C09102=1034.938,414.439,357.074,174.357,46.564,159.418
C09103=1034.949,414.684,357.028,174.369,46.569,159.421
C09104=1034.959,414.930,356.980,174.380,46.574,159.424
C09105=1034.970,415.176,356.933,174.392,46.580,159.427
C09106=1034.981,415.420,356.886,174.403,46.585,159.430
C09107=1034.991,415.666,356.839,174.415,46.591,159.433
C09108=1035.002,415.911,356.792,174.426,46.596,159.436
C09109=1035.013,416.157,356.745,174.438,46.602,159.439
C09110=1035.025,416.402,356.697,174.450,46.607,159.441
C09111=1035.035,416.647,356.650,174.461,46.613,159.444
C09112=1035.046,416.893,356.603,174.473,46.618,159.447
C09113=1035.057,417.137,356.555,174.485,46.623,159.450
C09114=1035.068,417.383,356.507,174.497,46.629,159.453
C09115=1035.078,417.628,356.459,174.509,46.635,159.456
C09116=1035.090,417.874,356.412,174.521,46.640,159.459
C09117=1035.100,418.118,356.364,174.533,46.646,159.462
C09118=1035.111,418.364,356.316,174.545,46.651,159.465
C09119=1035.121,418.609,356.269,174.556,46.657,159.468
C09120=1035.132,418.854,356.221,174.568,46.663,159.471
C09121=1035.144,419.100,356.172,174.581,46.668,159.474
C09122=1035.155,419.344,356.125,174.593,46.674,159.477
C09123=1035.166,419.589,356.077,174.605,46.680,159.480
C09124=1035.177,419.835,356.028,174.618,46.685,159.484
C09125=1035.187,420.079,355.980,174.630,46.691,159.487
C09126=1035.199,420.325,355.932,174.642,46.697,159.490
C09127=1035.210,420.570,355.884,174.655,46.703,159.493
C09128=1035.222,420.815,355.836,174.667,46.709,159.496
C09129=1035.233,421.061,355.788,174.679,46.714,159.499
C09130=1035.243,421.305,355.740,174.692,46.720,159.502
C09131=1035.255,421.550,355.691,174.704,46.726,159.506
C09132=1035.266,421.795,355.643,174.717,46.732,159.509
C09133=1035.277,422.041,355.594,174.729,46.738,159.512
C09134=1035.288,422.286,355.545,174.742,46.744,159.515
C09135=1035.300,422.531,355.498,174.754,46.750,159.518
C09136=1035.311,422.775,355.449,174.767,46.756,159.522
C09137=1035.323,423.021,355.400,174.780,46.762,159.525
C09138=1035.334,423.266,355.351,174.793,46.768,159.528
C09139=1035.346,423.511,355.303,174.805,46.774,159.531
C09140=1035.357,423.756,355.254,174.818,46.780,159.535
C09141=1035.368,424.001,355.205,174.832,46.786,159.538
C09142=1035.380,424.246,355.156,174.844,46.792,159.541
C09143=1035.391,424.490,355.107,174.857,46.798,159.545
C09144=1035.403,424.735,355.058,174.871,46.804,159.548
C09145=1035.414,424.982,355.008,174.883,46.810,159.551
C09146=1035.425,425.226,354.959,174.896,46.817,159.555
C09147=1035.437,425.470,354.910,174.910,46.823,159.558
C09148=1035.448,425.715,354.861,174.923,46.829,159.561
C09149=1035.460,425.961,354.811,174.936,46.835,159.565
C09150=1035.471,426.205,354.762,174.949,46.842,159.568
C09151=1035.483,426.450,354.713,174.963,46.848,159.572
C09152=1035.495,426.695,354.663,174.976,46.854,159.575
C09153=1035.507,426.940,354.614,174.990,46.861,159.579
C09154=1035.519,427.185,354.565,175.003,46.867,159.582
C09155=1035.530,427.429,354.515,175.016,46.873,159.585
C09156=1035.542,427.675,354.465,175.030,46.879,159.589
C09157=1035.553,427.919,354.415,175.043,46.886,159.593
C09158=1035.566,428.164,354.365,175.057,46.892,159.596
C09159=1035.577,428.408,354.315,175.071,46.899,159.600
C09160=1035.589,428.654,354.265,175.084,46.905,159.603
C09161=1035.600,428.898,354.216,175.099,46.912,159.607
C09162=1035.612,429.143,354.165,175.113,46.919,159.610
C09163=1035.624,429.387,354.115,175.127,46.925,159.614
C09164=1035.636,429.632,354.065,175.141,46.931,159.618
C09165=1035.647,429.877,354.014,175.154,46.939,159.621
C09166=1035.659,430.121,353.965,175.168,46.945,159.625
C09167=1035.672,430.366,353.915,175.182,46.952,159.629
C09168=1035.683,430.611,353.863,175.196,46.958,159.632
C09169=1035.696,430.855,353.813,175.211,46.965,159.636
C09170=1035.708,431.100,353.763,175.225,46.972,159.640
C09171=1035.719,431.345,353.713,175.239,46.979,159.644
C09172=1035.732,431.589,353.662,175.254,46.985,159.647
C09173=1035.744,431.834,353.612,175.268,46.992,159.651
C09174=1035.757,432.078,353.561,175.282,46.999,159.655
C09175=1035.768,432.323,353.510,175.297,47.005,159.659
C09176=1035.781,432.567,353.459,175.312,47.012,159.663
C09177=1035.793,432.811,353.409,175.326,47.019,159.666
C09178=1035.805,433.057,353.358,175.341,47.026,159.670
C09179=1035.818,433.301,353.307,175.355,47.033,159.674
C09180=1035.830,433.545,353.256,175.371,47.040,159.678
C09181=1035.842,433.789,353.205,175.385,47.047,159.682
C09182=1035.855,434.034,353.154,175.400,47.054,159.686
C09183=1035.867,434.279,353.102,175.415,47.060,159.690
C09184=1035.880,434.523,353.052,175.430,47.068,159.694
C09185=1035.893,434.768,353.000,175.445,47.074,159.697
C09186=1035.905,435.013,352.949,175.460,47.082,159.701
C09187=1035.917,435.257,352.898,175.475,47.089,159.705
C09188=1035.930,435.501,352.846,175.490,47.096,159.709
C09189=1035.942,435.746,352.794,175.505,47.103,159.713
C09190=1035.955,435.990,352.743,175.521,47.110,159.717
C09191=1035.967,436.234,352.691,175.537,47.117,159.721
C09192=1035.980,436.479,352.640,175.552,47.125,159.726
C09193=1035.993,436.725,352.588,175.567,47.132,159.730
C09194=1036.006,436.971,352.535,175.583,47.139,159.734
C09195=1036.018,437.216,352.484,175.598,47.147,159.738
C09196=1036.031,437.462,352.431,175.614,47.154,159.742
C09197=1036.044,437.707,352.379,175.630,47.161,159.746
C09198=1036.057,437.951,352.326,175.646,47.169,159.751
C09199=1036.070,438.195,352.275,175.662,47.176,159.755
C09200=1036.082,438.440,352.222,175.677,47.184,159.759
C09201=1036.095,438.683,352.170,175.693,47.191,159.763
C09202=1036.108,438.928,352.118,175.709,47.198,159.767
C09203=1036.121,439.172,352.066,175.725,47.206,159.772
C09204=1036.134,439.417,352.013,175.741,47.214,159.776
C09205=1036.147,439.660,351.961,175.757,47.221,159.780
C09206=1036.160,439.904,351.909,175.773,47.228,159.785
C09207=1036.173,440.148,351.855,175.789,47.236,159.789
C09208=1036.186,440.393,351.804,175.807,47.243,159.793
C09209=1036.199,440.637,351.750,175.823,47.251,159.798
C09210=1036.212,440.881,351.698,175.839,47.259,159.802
C09211=1036.225,441.125,351.645,175.856,47.267,159.807
C09212=1036.238,441.369,351.592,175.872,47.274,159.811
C09213=1036.252,441.613,351.539,175.889,47.282,159.816
C09214=1036.265,441.857,351.486,175.906,47.290,159.820
C09215=1036.278,442.101,351.432,175.922,47.297,159.825
C09216=1036.292,442.345,351.379,175.940,47.305,159.829
C09217=1036.305,442.588,351.327,175.956,47.313,159.834
C09218=1036.319,442.832,351.273,175.973,47.320,159.838
C09219=1036.332,443.076,351.220,175.990,47.329,159.843
C09220=1036.345,443.320,351.167,176.008,47.336,159.847
C09221=1036.359,443.563,351.114,176.024,47.344,159.852
C09222=1036.372,443.807,351.061,176.042,47.352,159.857
C09223=1036.386,444.050,351.007,176.058,47.360,159.861
C09224=1036.399,444.294,350.954,176.076,47.368,159.866
C09225=1036.414,444.537,350.901,176.094,47.376,159.870
C09226=1036.429,444.780,350.850,176.111,47.384,159.875
C09227=1036.445,445.024,350.797,176.129,47.391,159.880
C09228=1036.461,445.267,350.746,176.146,47.399,159.884
C09229=1036.478,445.511,350.695,176.164,47.406,159.889
C09230=1036.495,445.755,350.645,176.182,47.413,159.893
C09231=1036.513,445.999,350.595,176.200,47.421,159.898
C09232=1036.531,446.243,350.545,176.218,47.428,159.903
C09233=1036.550,446.486,350.497,176.236,47.435,159.907
C09234=1036.569,446.731,350.447,176.254,47.442,159.911
C09235=1036.589,446.975,350.399,176.272,47.449,159.916
C09236=1036.609,447.220,350.351,176.291,47.456,159.921
C09237=1036.630,447.464,350.304,176.309,47.462,159.925
C09238=1036.652,447.708,350.257,176.327,47.469,159.929
C09239=1036.673,447.953,350.211,176.346,47.475,159.934
C09240=1036.697,448.198,350.165,176.364,47.482,159.938
C09241=1036.719,448.442,350.119,176.383,47.488,159.943
C09242=1036.743,448.687,350.074,176.401,47.495,159.947
C09243=1036.767,448.931,350.029,176.421,47.501,159.952
C09244=1036.792,449.177,349.985,176.440,47.507,159.956
C09245=1036.817,449.422,349.941,176.459,47.513,159.961
C09246=1036.843,449.667,349.898,176.478,47.519,159.965
C09247=1036.869,449.912,349.855,176.497,47.525,159.969
C09248=1036.896,450.157,349.812,176.517,47.530,159.974
C09249=1036.924,450.403,349.771,176.536,47.536,159.978
C09250=1036.951,450.649,349.729,176.555,47.541,159.982
C09251=1036.980,450.893,349.687,176.575,47.548,159.987
C09252=1037.009,451.139,349.647,176.594,47.553,159.991
C09253=1037.046,451.441,349.597,176.619,47.560,159.996
C09254=1037.083,451.744,349.549,176.644,47.566,160.002
C09255=1037.122,452.046,349.501,176.668,47.572,160.007
C09256=1037.160,452.347,349.453,176.693,47.578,160.012
C09257=1036.869,452.403,349.129,176.696,47.649,160.034
C09258=1036.832,452.115,349.174,176.672,47.644,160.029
C09259=1036.796,451.826,349.221,176.648,47.637,160.024
C09260=1036.760,451.537,349.267,176.625,47.632,160.019
C09261=1036.724,451.248,349.314,176.602,47.626,160.014
C09262=1036.695,451.003,349.354,176.582,47.620,160.010
C09263=1036.666,450.758,349.395,176.562,47.615,160.006
C09264=1036.638,450.512,349.436,176.543,47.609,160.001
C09265=1036.610,450.266,349.478,176.523,47.604,159.997
C09266=1036.583,450.021,349.520,176.504,47.598,159.992
C09267=1036.557,449.776,349.563,176.484,47.592,159.988
C09268=1036.531,449.531,349.606,176.465,47.586,159.984
C09269=1036.504,449.286,349.650,176.446,47.580,159.979
C09270=1036.480,449.041,349.693,176.427,47.574,159.975
C09271=1036.455,448.796,349.739,176.408,47.569,159.971
C09272=1036.431,448.551,349.783,176.389,47.562,159.966
C09273=1036.407,448.306,349.829,176.371,47.556,159.962
C09274=1036.385,448.062,349.874,176.351,47.549,159.957
C09275=1036.363,447.816,349.920,176.333,47.543,159.953
C09276=1036.341,447.572,349.967,176.314,47.537,159.948
C09277=1036.319,447.328,350.014,176.296,47.530,159.944
C09278=1036.298,447.084,350.062,176.278,47.523,159.939
C09279=1036.279,446.839,350.110,176.259,47.517,159.935
C09280=1036.259,446.595,350.159,176.241,47.510,159.930
C09281=1036.240,446.351,350.206,176.223,47.503,159.926
C09282=1036.221,446.107,350.256,176.204,47.496,159.921
C09283=1036.203,445.863,350.306,176.187,47.489,159.917
C09284=1036.185,445.619,350.356,176.168,47.482,159.912
C09285=1036.169,445.375,350.407,176.151,47.474,159.908
C09286=1036.152,445.132,350.458,176.133,47.467,159.903
C09287=1036.137,444.888,350.509,176.116,47.459,159.898
C09288=1036.121,444.645,350.561,176.098,47.452,159.894
C09289=1036.106,444.402,350.613,176.081,47.444,159.889
C09290=1036.092,444.159,350.667,176.063,47.437,159.885
C09291=1036.078,443.915,350.719,176.046,47.429,159.880
C09292=1036.065,443.672,350.773,176.029,47.421,159.875
C09293=1036.051,443.429,350.827,176.011,47.413,159.871
C09294=1036.038,443.185,350.880,175.994,47.405,159.866
C09295=1036.025,442.941,350.933,175.977,47.398,159.862
C09296=1036.011,442.697,350.986,175.960,47.390,159.857
C09297=1035.997,442.453,351.039,175.943,47.382,159.852
C09298=1035.984,442.209,351.093,175.926,47.375,159.848
C09299=1035.970,441.966,351.146,175.910,47.367,159.843
C09300=1035.957,441.721,351.198,175.892,47.359,159.839
C09301=1035.944,441.477,351.251,175.876,47.351,159.834
C09302=1035.931,441.233,351.305,175.859,47.344,159.830
C09303=1035.917,440.989,351.357,175.842,47.336,159.825
C09304=1035.904,440.745,351.410,175.826,47.328,159.821
C09305=1035.891,440.501,351.463,175.809,47.321,159.817
C09306=1035.878,440.257,351.516,175.793,47.314,159.812
C09307=1035.866,440.013,351.568,175.777,47.306,159.808
C09308=1035.852,439.769,351.621,175.761,47.298,159.804
C09309=1035.839,439.525,351.673,175.744,47.291,159.799
C09310=1035.826,439.281,351.727,175.728,47.284,159.795
C09311=1035.813,439.036,351.778,175.711,47.276,159.791
C09312=1035.800,438.793,351.831,175.695,47.269,159.786
C09313=1035.787,438.548,351.882,175.679,47.262,159.782
C09314=1035.774,438.304,351.935,175.664,47.255,159.778
C09315=1035.762,438.060,351.987,175.648,47.247,159.774
C09316=1035.748,437.815,352.039,175.632,47.239,159.769
C09317=1035.736,437.571,352.091,175.617,47.233,159.765
C09318=1035.723,437.324,352.145,175.600,47.225,159.761
C09319=1035.710,437.076,352.197,175.584,47.218,159.757
C09320=1035.697,436.829,352.249,175.569,47.211,159.753
C09321=1035.684,436.582,352.302,175.553,47.203,159.749
C09322=1035.672,436.338,352.353,175.538,47.196,159.745
C09323=1035.659,436.094,352.405,175.522,47.189,159.740
C09324=1035.646,435.849,352.457,175.506,47.182,159.736
C09325=1035.634,435.605,352.508,175.492,47.175,159.732
C09326=1035.622,435.361,352.559,175.476,47.168,159.728
C09327=1035.608,435.116,352.611,175.461,47.161,159.724
C09328=1035.596,434.872,352.663,175.446,47.154,159.720
C09329=1035.584,434.628,352.714,175.431,47.147,159.716
C09330=1035.572,434.383,352.765,175.415,47.140,159.712
C09331=1035.559,434.138,352.816,175.401,47.133,159.709
C09332=1035.547,433.894,352.868,175.387,47.126,159.705
C09333=1035.534,433.650,352.918,175.371,47.119,159.701
C09334=1035.522,433.405,352.968,175.356,47.112,159.697
C09335=1035.510,433.160,353.020,175.341,47.106,159.693
C09336=1035.497,432.915,353.071,175.326,47.099,159.689
C09337=1035.484,432.671,353.122,175.312,47.092,159.685
C09338=1035.472,432.426,353.173,175.298,47.085,159.681
C09339=1035.460,432.182,353.223,175.283,47.078,159.678
C09340=1035.447,431.938,353.274,175.268,47.072,159.674
C09341=1035.435,431.694,353.324,175.254,47.065,159.670
C09342=1035.424,431.448,353.375,175.239,47.059,159.666
C09343=1035.411,431.204,353.425,175.225,47.052,159.663
C09344=1035.399,430.959,353.476,175.211,47.045,159.659
C09345=1035.387,430.714,353.526,175.197,47.039,159.655
C09346=1035.375,430.470,353.577,175.182,47.032,159.651
C09347=1035.363,430.226,353.627,175.168,47.025,159.648
C09348=1035.351,429.981,353.677,175.154,47.019,159.644
C09349=1035.339,429.736,353.728,175.140,47.012,159.641
C09350=1035.327,429.491,353.778,175.126,47.006,159.637
C09351=1035.316,429.247,353.828,175.112,47.000,159.633
C09352=1035.304,429.002,353.878,175.098,46.992,159.630
C09353=1035.292,428.758,353.928,175.084,46.986,159.626
C09354=1035.280,428.513,353.978,175.070,46.980,159.622
C09355=1035.269,428.268,354.028,175.056,46.973,159.619
C09356=1035.257,428.023,354.078,175.042,46.967,159.615
C09357=1035.245,427.779,354.127,175.029,46.960,159.612
C09358=1035.233,427.534,354.178,175.016,46.955,159.608
C09359=1035.222,427.289,354.227,175.002,46.948,159.605
C09360=1035.210,427.044,354.277,174.989,46.942,159.601
C09361=1035.198,426.799,354.326,174.975,46.936,159.598
C09362=1035.186,426.554,354.375,174.961,46.929,159.594
C09363=1035.174,426.310,354.425,174.948,46.923,159.591
C09364=1035.162,426.064,354.475,174.934,46.917,159.587
C09365=1035.151,425.820,354.524,174.921,46.911,159.584
C09366=1035.140,425.575,354.573,174.907,46.904,159.581
C09367=1035.128,425.329,354.623,174.895,46.898,159.577
C09368=1035.117,425.085,354.672,174.881,46.892,159.574
C09369=1035.105,424.840,354.721,174.868,46.886,159.571
C09370=1035.094,424.596,354.770,174.856,46.880,159.567
C09371=1035.083,424.350,354.819,174.842,46.874,159.564
C09372=1035.071,424.105,354.868,174.829,46.868,159.561
C09373=1035.059,423.860,354.917,174.816,46.862,159.557
C09374=1035.048,423.615,354.966,174.803,46.856,159.554
C09375=1035.037,423.371,355.015,174.790,46.850,159.551
C09376=1035.025,423.125,355.063,174.778,46.844,159.548
C09377=1035.014,422.880,355.112,174.764,46.838,159.544
C09378=1035.003,422.633,355.161,174.752,46.832,159.541
C09379=1034.990,422.386,355.210,174.739,46.826,159.538
C09380=1034.979,422.138,355.259,174.726,46.821,159.534
C09381=1034.968,421.890,355.308,174.713,46.814,159.531
C09382=1034.957,421.645,355.356,174.701,46.809,159.528
C09383=1034.945,421.400,355.405,174.688,46.803,159.525
C09384=1034.934,421.155,355.453,174.676,46.797,159.522
C09385=1034.923,420.910,355.501,174.663,46.791,159.519
C09386=1034.912,420.665,355.549,174.651,46.786,159.515
C09387=1034.901,420.421,355.598,174.639,46.780,159.512
C09388=1034.890,420.175,355.647,174.626,46.774,159.509
C09389=1034.878,419.930,355.695,174.614,46.769,159.506
C09390=1034.867,419.685,355.742,174.602,46.763,159.503
C09391=1034.856,419.440,355.791,174.590,46.757,159.500
C09392=1034.845,419.194,355.838,174.577,46.752,159.497
C09393=1034.834,418.949,355.887,174.565,46.746,159.494
C09394=1034.824,418.704,355.934,174.553,46.740,159.491
C09395=1034.813,418.459,355.983,174.541,46.735,159.488
C09396=1034.801,418.214,356.030,174.528,46.729,159.485
C09397=1034.791,417.968,356.078,174.517,46.723,159.482
C09398=1034.780,417.724,356.126,174.505,46.718,159.479
C09399=1034.769,417.478,356.174,174.493,46.712,159.476
C09400=1034.759,417.233,356.221,174.481,46.707,159.473
C09401=1034.747,416.988,356.269,174.468,46.702,159.470
C09402=1034.737,416.743,356.316,174.457,46.696,159.467
C09403=1034.725,416.497,356.363,174.445,46.691,159.464
C09404=1034.715,416.252,356.411,174.433,46.686,159.461
C09405=1034.703,416.007,356.458,174.422,46.680,159.458
C09406=1034.693,415.761,356.505,174.410,46.675,159.455
C09407=1034.682,415.515,356.553,174.398,46.669,159.452
C09408=1034.671,415.271,356.599,174.387,46.664,159.449
C09409=1034.661,415.025,356.647,174.375,46.659,159.446
C09410=1034.650,414.780,356.694,174.363,46.654,159.444
C09411=1034.639,414.535,356.741,174.352,46.648,159.441
C09412=1034.628,414.289,356.787,174.340,46.643,159.438
C09413=1034.618,414.044,356.835,174.330,46.638,159.435
C09414=1034.607,413.799,356.881,174.318,46.633,159.432
C09415=1034.597,413.553,356.929,174.307,46.627,159.430
C09416=1034.586,413.308,356.975,174.295,46.623,159.427
C09417=1034.575,413.063,357.023,174.284,46.617,159.424
C09418=1034.566,412.817,357.069,174.272,46.612,159.421
C09419=1034.555,412.572,357.116,174.261,46.607,159.419
C09420=1034.544,412.327,357.163,174.250,46.602,159.416
C09421=1034.534,412.081,357.209,174.239,46.597,159.413
C09422=1034.524,411.836,357.256,174.228,46.591,159.410
C09423=1034.513,411.590,357.302,174.217,46.586,159.408
C09424=1034.503,411.345,357.349,174.205,46.582,159.405
C09425=1034.492,411.099,357.395,174.194,46.576,159.402
C09426=1034.482,410.854,357.442,174.184,46.571,159.399
C09427=1034.471,410.608,357.488,174.172,46.567,159.397
C09428=1034.461,410.363,357.534,174.162,46.562,159.394
C09429=1034.450,410.117,357.580,174.151,46.557,159.391
C09430=1034.440,409.871,357.627,174.140,46.552,159.389
C09431=1034.430,409.626,357.672,174.129,46.547,159.386
C09432=1034.419,409.381,357.719,174.118,46.542,159.384
C09433=1034.408,409.135,357.765,174.108,46.538,159.381
C09434=1034.398,408.893,357.810,174.097,46.533,159.378
C09435=1034.389,408.651,357.855,174.086,46.528,159.376
C09436=1034.378,408.410,357.900,174.076,46.523,159.373
C09437=1034.367,408.168,357.946,174.065,46.518,159.371
C09438=1034.358,407.926,357.990,174.055,46.514,159.368
C09439=1034.347,407.685,358.036,174.044,46.509,159.366
C09440=1034.338,407.443,358.081,174.034,46.504,159.363
C09441=1034.328,407.201,358.126,174.024,46.500,159.361
C09442=1034.317,406.955,358.172,174.013,46.495,159.358
C09443=1034.308,406.710,358.216,174.003,46.491,159.356
C09444=1034.297,406.464,358.262,173.992,46.486,159.353
C09445=1034.287,406.219,358.308,173.982,46.481,159.351
C09446=1034.277,405.973,358.354,173.972,46.477,159.348
C09447=1034.267,405.728,358.399,173.961,46.472,159.346
C09448=1034.257,405.482,358.444,173.951,46.467,159.343
C09449=1034.247,405.237,358.490,173.940,46.463,159.341
C09450=1034.237,404.991,358.535,173.930,46.458,159.339
C09451=1034.228,404.745,358.581,173.920,46.454,159.336
C09452=1034.217,404.499,358.626,173.909,46.449,159.333
C09453=1034.207,404.254,358.671,173.900,46.444,159.331
C09454=1034.198,404.008,358.716,173.889,46.440,159.329
C09455=1034.187,403.763,358.762,173.879,46.435,159.326
C09456=1034.177,403.517,358.807,173.869,46.431,159.324
C09457=1034.168,403.271,358.852,173.859,46.427,159.322
C09458=1034.158,403.025,358.897,173.850,46.422,159.319
C09459=1034.148,402.779,358.942,173.839,46.418,159.317
C09460=1034.139,402.534,358.987,173.829,46.413,159.314
C09461=1034.129,402.288,359.032,173.819,46.409,159.312
C09462=1034.118,402.042,359.077,173.809,46.405,159.310
C09463=1034.109,401.797,359.122,173.799,46.400,159.307
C09464=1034.099,401.551,359.167,173.789,46.395,159.305
C09465=1034.089,401.306,359.212,173.779,46.391,159.303
C09466=1034.080,401.060,359.256,173.770,46.387,159.300
C09467=1034.070,400.814,359.301,173.760,46.383,159.298
C09468=1034.060,400.568,359.346,173.749,46.378,159.296
C09469=1034.050,400.322,359.390,173.740,46.374,159.294
C09470=1034.040,400.077,359.434,173.730,46.370,159.291
C09471=1034.030,399.831,359.479,173.720,46.366,159.289
C09472=1034.021,399.585,359.523,173.711,46.361,159.287
C09473=1034.011,399.339,359.568,173.701,46.358,159.285
C09474=1034.002,399.093,359.612,173.692,46.353,159.282
C09475=1033.992,398.847,359.656,173.682,46.349,159.280
C09476=1033.982,398.602,359.700,173.672,46.345,159.278
C09477=1033.973,398.356,359.744,173.663,46.341,159.276
C09478=1033.963,398.110,359.788,173.653,46.337,159.273
C09479=1033.953,397.864,359.833,173.644,46.332,159.271
C09480=1033.944,397.619,359.876,173.634,46.328,159.269
C09481=1033.934,397.373,359.921,173.625,46.324,159.267
C09482=1033.925,397.145,359.962,173.616,46.321,159.265
C09483=1033.917,396.916,360.002,173.608,46.317,159.263
C09484=1033.908,396.687,360.044,173.599,46.313,159.261
C09485=1033.899,396.460,360.084,173.590,46.310,159.259
C09486=1033.890,396.231,360.124,173.582,46.306,159.257
C09487=1033.881,396.003,360.166,173.573,46.302,159.255
C09488=1033.873,395.775,360.207,173.564,46.299,159.253
C09489=1033.863,395.546,360.246,173.556,46.295,159.251
C09490=1033.854,395.300,360.291,173.547,46.291,159.249
C09491=1033.845,395.055,360.334,173.537,46.287,159.247
C09492=1033.836,394.809,360.378,173.528,46.283,159.245
C09493=1033.826,394.563,360.422,173.519,46.279,159.243
C09494=1033.817,394.317,360.465,173.509,46.276,159.241
C09495=1033.808,394.071,360.509,173.500,46.271,159.238
C09496=1033.798,393.825,360.553,173.492,46.268,159.236
C09497=1033.789,393.579,360.596,173.482,46.264,159.234
C09498=1033.779,393.327,360.641,173.473,46.260,159.232
C09499=1033.769,393.074,360.685,173.463,46.256,159.230
C09500=1033.760,392.822,360.729,173.454,46.252,159.228
C09501=1033.750,392.570,360.774,173.445,46.248,159.226
C09502=1033.741,392.324,360.817,173.436,46.245,159.224
C09503=1033.732,392.078,360.860,173.427,46.241,159.222
C09504=1033.722,391.832,360.903,173.419,46.237,159.220
C09505=1033.713,391.586,360.947,173.410,46.233,159.218
C09506=1033.704,391.340,360.989,173.400,46.230,159.216
C09507=1033.695,391.093,361.033,173.391,46.226,159.214
C09508=1033.685,390.848,361.076,173.383,46.222,159.212
C09509=1033.677,390.602,361.119,173.374,46.218,159.210
C09510=1033.667,390.356,361.162,173.365,46.215,159.208
C09511=1033.658,390.110,361.205,173.357,46.212,159.206
C09512=1033.648,389.863,361.247,173.347,46.208,159.204
C09513=1033.639,389.617,361.290,173.339,46.204,159.202
C09514=1033.631,389.371,361.333,173.330,46.201,159.200
C09515=1033.621,389.125,361.376,173.321,46.197,159.198
C09516=1033.612,388.879,361.419,173.313,46.194,159.197
C09517=1033.603,388.633,361.461,173.304,46.190,159.195
C09518=1033.594,388.387,361.504,173.296,46.186,159.193
C09519=1033.585,388.141,361.547,173.287,46.183,159.191
C09520=1033.575,387.895,361.589,173.279,46.180,159.189
C09521=1033.567,387.648,361.631,173.270,46.176,159.187
C09522=1033.558,387.402,361.674,173.262,46.173,159.185
C09523=1033.548,387.156,361.717,173.253,46.169,159.183
C09524=1033.539,386.910,361.759,173.245,46.166,159.181
C09525=1033.530,386.664,361.801,173.236,46.162,159.179
C09526=1033.521,386.418,361.844,173.228,46.159,159.178
C09527=1033.512,386.172,361.885,173.219,46.156,159.176
C09528=1033.503,385.925,361.929,173.211,46.152,159.174
C09529=1033.494,385.679,361.970,173.202,46.149,159.172
C09530=1033.485,385.433,362.013,173.194,46.146,159.170
C09531=1033.476,385.187,362.055,173.186,46.143,159.169
C09532=1033.467,384.940,362.096,173.177,46.139,159.167
C09533=1033.457,384.694,362.139,173.169,46.136,159.165
C09534=1033.449,384.448,362.180,173.160,46.132,159.163
C09535=1033.440,384.202,362.222,173.152,46.129,159.161
C09536=1033.431,383.955,362.264,173.144,46.126,159.160
C09537=1033.421,383.710,362.306,173.135,46.123,159.158
C09538=1033.412,383.463,362.348,173.128,46.120,159.156
C09539=1033.404,383.217,362.390,173.120,46.116,159.154
C09540=1033.395,382.970,362.432,173.111,46.113,159.153
C09541=1033.386,382.724,362.474,173.103,46.110,159.151
C09542=1033.377,382.477,362.515,173.095,46.107,159.149
C09543=1033.369,382.231,362.557,173.086,46.104,159.147
C09544=1033.360,381.985,362.599,173.079,46.100,159.146
C09545=1033.351,381.738,362.641,173.070,46.097,159.144
C09546=1033.342,381.493,362.682,173.062,46.094,159.142
C09547=1033.333,381.246,362.724,173.054,46.091,159.140
C09548=1033.324,381.000,362.765,173.046,46.088,159.139
C09549=1033.316,380.754,362.807,173.038,46.085,159.137
C09550=1033.307,380.507,362.849,173.030,46.082,159.135
C09551=1033.298,380.261,362.891,173.022,46.079,159.134
C09552=1033.289,380.015,362.932,173.015,46.075,159.132
C09553=1033.281,379.768,362.973,173.006,46.072,159.130
C09554=1033.274,379.554,363.009,173.000,46.070,159.129
C09555=1033.266,379.341,363.045,172.993,46.067,159.127
C09556=1033.259,379.126,363.082,172.986,46.065,159.126
C09557=1033.251,378.912,363.117,172.979,46.062,159.124
C09558=1033.244,378.698,363.153,172.972,46.060,159.123
C09559=1033.236,378.484,363.189,172.965,46.057,159.122
C09560=1033.229,378.270,363.226,172.958,46.055,159.120
C09561=1033.221,378.056,363.261,172.952,46.051,159.119
C09562=1033.213,377.810,363.302,172.944,46.049,159.117
C09563=1033.204,377.563,363.343,172.936,46.046,159.115
C09564=1033.196,377.316,363.384,172.929,46.043,159.114
C09565=1033.187,377.071,363.425,172.921,46.040,159.112
C09566=1033.178,376.824,363.466,172.913,46.038,159.111
C09567=1033.169,376.577,363.507,172.905,46.034,159.109
C09568=1033.161,376.331,363.548,172.897,46.031,159.107
C09569=1033.152,376.085,363.589,172.890,46.029,159.106
C09570=1033.144,375.838,363.629,172.882,46.026,159.104
C09571=1033.135,375.591,363.670,172.874,46.023,159.103
C09572=1033.126,375.345,363.710,172.867,46.020,159.101
C09573=1033.118,375.098,363.751,172.859,46.018,159.100
C09574=1033.110,374.852,363.792,172.852,46.015,159.098
C09575=1033.101,374.606,363.834,172.844,46.012,159.097
C09576=1033.092,374.360,363.874,172.837,46.009,159.095
C09577=1033.083,374.113,363.915,172.829,46.007,159.094
C09578=1033.075,373.867,363.956,172.822,46.004,159.092
C09579=1033.066,373.620,363.996,172.814,46.001,159.090
C09580=1033.058,373.373,364.036,172.807,45.998,159.089
C09581=1033.050,373.127,364.076,172.799,45.996,159.087
C09582=1033.041,372.880,364.117,172.792,45.993,159.086
C09583=1033.033,372.634,364.158,172.784,45.990,159.084
C09584=1033.024,372.387,364.199,172.777,45.987,159.083
C09585=1033.016,372.140,364.239,172.769,45.985,159.081
C09586=1033.008,371.894,364.278,172.762,45.982,159.080
C09587=1032.999,371.647,364.319,172.755,45.979,159.078
C09588=1032.991,371.401,364.360,172.747,45.977,159.077
C09589=1032.982,371.155,364.400,172.740,45.974,159.075
C09590=1032.974,370.908,364.440,172.732,45.972,159.074
C09591=1032.966,370.661,364.481,172.725,45.969,159.072
C09592=1032.958,370.414,364.522,172.718,45.967,159.071
C09593=1032.949,370.168,364.561,172.710,45.964,159.069
C09594=1032.941,369.922,364.602,172.704,45.962,159.068
C09595=1032.934,369.675,364.642,172.697,45.959,159.067
C09596=1032.924,369.428,364.682,172.689,45.957,159.065
C09597=1032.916,369.181,364.722,172.682,45.954,159.064
C09598=1032.908,368.935,364.761,172.675,45.951,159.062
C09599=1032.899,368.689,364.801,172.667,45.949,159.061
C09600=1032.892,368.442,364.841,172.660,45.946,159.059
C09601=1032.882,368.194,364.881,172.654,45.944,159.058
C09602=1032.874,367.948,364.920,172.646,45.942,159.057
C09603=1032.866,367.701,364.961,172.639,45.939,159.055
C09604=1032.858,367.455,365.000,172.632,45.937,159.054
C09605=1032.849,367.208,365.039,172.624,45.935,159.052
C09606=1032.841,366.961,365.079,172.618,45.932,159.051
C09607=1032.833,366.715,365.119,172.611,45.929,159.050
C09608=1032.825,366.468,365.159,172.604,45.927,159.048
C09609=1032.817,366.221,365.198,172.596,45.925,159.047
C09610=1032.808,365.975,365.238,172.590,45.923,159.046
C09611=1032.800,365.728,365.278,172.583,45.920,159.044
C09612=1032.792,365.482,365.317,172.576,45.918,159.043
C09613=1032.784,365.235,365.356,172.568,45.916,159.041
C09614=1032.770,364.828,365.422,172.557,45.912,159.039
C09615=1032.756,364.420,365.487,172.546,45.908,159.037
C09616=1032.743,364.013,365.552,172.535,45.904,159.035
C09617=1032.730,363.606,365.617,172.523,45.900,159.033
C09618=1032.722,363.359,365.656,172.516,45.898,159.031
C09619=1032.713,363.113,365.695,172.510,45.896,159.030
C09620=1032.706,362.865,365.735,172.503,45.894,159.029
C09621=1032.697,362.618,365.774,172.496,45.892,159.027
C09622=1032.690,362.373,365.813,172.488,45.890,159.026
C09623=1032.682,362.125,365.852,172.482,45.887,159.025
C09624=1032.674,361.878,365.891,172.475,45.885,159.023
C09625=1032.665,361.632,365.931,172.469,45.883,159.022
C09626=1032.658,361.384,365.970,172.462,45.881,159.021
C09627=1032.650,361.138,366.009,172.455,45.878,159.020
C09628=1032.642,360.891,366.048,172.449,45.877,159.018
C09629=1032.633,360.645,366.087,172.442,45.874,159.017
C09630=1032.625,360.397,366.125,172.435,45.872,159.016
C09631=1032.618,360.151,366.164,172.429,45.870,159.015
C09632=1032.609,359.904,366.203,172.422,45.868,159.013
C09633=1032.601,359.657,366.242,172.415,45.866,159.012
C09634=1032.594,359.410,366.281,172.408,45.864,159.011
C09635=1032.586,359.164,366.320,172.401,45.862,159.010
C09636=1032.578,358.916,366.358,172.395,45.860,159.008
C09637=1032.569,358.669,366.397,172.388,45.858,159.007
C09638=1032.562,358.423,366.435,172.382,45.856,159.006
C09639=1032.553,358.176,366.475,172.375,45.854,159.005
C09640=1032.545,357.929,366.513,172.369,45.852,159.004
C09641=1032.538,357.682,366.551,172.362,45.850,159.002
C09642=1032.530,357.435,366.590,172.356,45.848,159.001
C09643=1032.521,357.188,366.629,172.349,45.846,159.000
C09644=1032.514,356.941,366.667,172.342,45.844,158.999
C09645=1032.506,356.694,366.706,172.336,45.842,158.997
C09646=1032.498,356.448,366.744,172.329,45.840,158.996
C09647=1032.490,356.200,366.782,172.323,45.839,158.995
C09648=1032.483,355.954,366.821,172.316,45.836,158.994
C09649=1032.474,355.707,366.859,172.310,45.834,158.993
C09650=1032.466,355.460,366.898,172.303,45.833,158.992
C09651=1032.459,355.213,366.936,172.297,45.831,158.990
C09652=1032.450,354.965,366.973,172.292,45.829,158.989
C09653=1032.443,354.719,367.012,172.285,45.827,158.988
C09654=1032.434,354.472,367.050,172.279,45.825,158.987
C09655=1032.427,354.225,367.088,172.272,45.824,158.986
C09656=1032.419,353.977,367.126,172.266,45.822,158.985
C09657=1032.411,353.731,367.164,172.259,45.820,158.984
C09658=1032.403,353.484,367.203,172.253,45.818,158.982
C09659=1032.395,353.237,367.240,172.247,45.816,158.981
C09660=1032.388,352.990,367.278,172.240,45.815,158.980
C09661=1032.380,352.743,367.317,172.234,45.813,158.979
C09662=1032.372,352.496,367.354,172.227,45.811,158.978
C09663=1032.363,352.249,367.393,172.222,45.809,158.977
C09664=1032.356,352.002,367.430,172.215,45.807,158.976
C09665=1032.349,351.755,367.468,172.209,45.806,158.974
C09666=1032.341,351.508,367.506,172.203,45.804,158.973
C09667=1032.333,351.261,367.544,172.196,45.803,158.972
C09668=1032.325,351.014,367.581,172.190,45.801,158.971
C09669=1032.317,350.767,367.620,172.185,45.799,158.970
C09670=1032.305,350.366,367.681,172.174,45.796,158.968
C09671=1032.293,349.965,367.742,172.164,45.794,158.967
C09672=1032.279,349.564,367.803,172.154,45.791,158.965
C09673=1032.267,349.163,367.865,172.144,45.788,158.963
C09674=1032.260,348.916,367.902,172.138,45.786,158.962
C09675=1032.253,348.669,367.940,172.132,45.785,158.961
C09676=1032.244,348.422,367.978,172.126,45.783,158.960
C09677=1032.237,348.175,368.015,172.119,45.782,158.959
C09678=1032.229,347.928,368.052,172.113,45.780,158.958
C09679=1032.221,347.681,368.090,172.108,45.778,158.957
C09680=1032.213,347.434,368.127,172.102,45.777,158.956
C09681=1032.206,347.186,368.164,172.095,45.775,158.955
C09682=1032.198,346.940,368.201,172.089,45.774,158.954
C09683=1032.190,346.692,368.239,172.084,45.772,158.953
C09684=1032.182,346.446,368.276,172.078,45.771,158.952
C09685=1032.175,346.198,368.313,172.071,45.769,158.950
C09686=1032.167,345.952,368.350,172.066,45.768,158.950
C09687=1032.160,345.705,368.388,172.060,45.767,158.949
C09688=1032.152,345.458,368.425,172.053,45.765,158.947
C09689=1032.144,345.209,368.462,172.047,45.764,158.946
C09690=1032.136,344.962,368.499,172.042,45.762,158.946
C09691=1032.129,344.715,368.536,172.036,45.760,158.944
C09692=1032.121,344.468,368.573,172.030,45.759,158.943
C09693=1032.114,344.221,368.611,172.024,45.758,158.943
C09694=1032.106,343.974,368.647,172.018,45.756,158.942
C09695=1032.099,343.727,368.685,172.012,45.755,158.940
C09696=1032.091,343.480,368.722,172.007,45.753,158.940
C09697=1032.084,343.232,368.758,172.001,45.752,158.939
C09698=1032.076,342.985,368.795,171.994,45.751,158.938
C09699=1032.069,342.738,368.833,171.989,45.749,158.937
C09700=1032.061,342.491,368.869,171.983,45.747,158.936
C09701=1032.053,342.244,368.906,171.977,45.746,158.935
C09702=1032.046,341.997,368.943,171.972,45.745,158.934
C09703=1032.038,341.749,368.980,171.965,45.744,158.933
C09704=1032.032,341.503,369.017,171.960,45.742,158.932
C09705=1032.024,341.255,369.053,171.954,45.741,158.931
C09706=1032.016,341.009,369.090,171.948,45.740,158.930
C09707=1032.009,340.761,369.127,171.943,45.738,158.929
C09708=1032.001,340.513,369.163,171.937,45.737,158.928
C09709=1031.993,340.267,369.200,171.932,45.736,158.927
C09710=1031.986,340.019,369.236,171.925,45.734,158.926
C09711=1031.979,339.771,369.273,171.919,45.733,158.925
C09712=1031.971,339.525,369.310,171.914,45.732,158.924
C09713=1031.964,339.278,369.346,171.908,45.730,158.923
C09714=1031.956,339.030,369.382,171.903,45.730,158.923
C09715=1031.948,338.783,369.418,171.897,45.728,158.922
C09716=1031.940,338.536,369.455,171.891,45.727,158.921
C09717=1031.933,338.288,369.492,171.886,45.726,158.920
C09718=1031.926,338.041,369.528,171.880,45.725,158.919
C09719=1031.919,337.794,369.564,171.875,45.724,158.918
C09720=1031.911,337.547,369.600,171.869,45.722,158.917
C09721=1031.903,337.299,369.636,171.863,45.721,158.916
C09722=1031.895,337.052,369.673,171.857,45.720,158.915
C09723=1031.889,336.805,369.710,171.852,45.719,158.914
C09724=1031.881,336.558,369.746,171.846,45.718,158.913
C09725=1031.874,336.311,369.782,171.841,45.716,158.913
C09726=1031.862,335.906,369.841,171.831,45.715,158.911
C09727=1031.850,335.502,369.901,171.823,45.713,158.910
C09728=1031.838,335.098,369.960,171.814,45.711,158.908
C09729=1031.826,334.694,370.019,171.804,45.709,158.907
C09730=1031.819,334.446,370.055,171.799,45.708,158.906
C09731=1031.811,334.199,370.091,171.793,45.707,158.905
C09732=1031.804,333.952,370.127,171.788,45.706,158.904
C09733=1031.796,333.704,370.162,171.782,45.705,158.903
C09734=1031.789,333.457,370.198,171.777,45.704,158.903
C09735=1031.781,333.210,370.234,171.771,45.703,158.902
C09736=1031.774,332.962,370.269,171.766,45.702,158.901
C09737=1031.766,332.715,370.305,171.762,45.701,158.900
C09738=1031.759,332.468,370.341,171.755,45.700,158.899
C09739=1031.752,332.220,370.376,171.751,45.699,158.899
C09740=1031.744,331.973,370.413,171.744,45.698,158.898
C09741=1031.737,331.725,370.449,171.740,45.697,158.897
C09742=1031.730,331.478,370.484,171.734,45.696,158.896
C09743=1031.722,331.231,370.520,171.729,45.695,158.895
C09744=1031.715,330.984,370.555,171.723,45.694,158.894
C09745=1031.707,330.736,370.591,171.718,45.693,158.894
C09746=1031.700,330.489,370.626,171.713,45.692,158.893
C09747=1031.693,330.241,370.662,171.707,45.691,158.892
C09748=1031.686,329.994,370.698,171.702,45.690,158.891
C09749=1031.678,329.746,370.734,171.696,45.690,158.890
C09750=1031.671,329.499,370.769,171.691,45.688,158.890
C09751=1031.664,329.252,370.805,171.686,45.687,158.889
C09752=1031.657,329.004,370.840,171.680,45.687,158.888
C09753=1031.649,328.758,370.875,171.675,45.686,158.887
C09754=1031.642,328.510,370.911,171.671,45.685,158.887
C09755=1031.635,328.262,370.946,171.664,45.684,158.886
C09756=1031.628,328.016,370.982,171.660,45.683,158.885
C09757=1031.621,327.768,371.017,171.655,45.682,158.884
C09758=1031.613,327.521,371.052,171.649,45.681,158.883
C09759=1031.606,327.273,371.088,171.644,45.680,158.883
C09760=1031.598,327.025,371.122,171.638,45.680,158.882
C09761=1031.590,326.778,371.157,171.633,45.679,158.881
C09762=1031.583,326.530,371.192,171.628,45.678,158.880
C09763=1031.576,326.283,371.227,171.622,45.677,158.880
C09764=1031.568,326.036,371.263,171.618,45.677,158.879
C09765=1031.561,325.789,371.297,171.612,45.676,158.878
C09766=1031.553,325.541,371.333,171.607,45.676,158.877
C09767=1031.546,325.294,371.367,171.602,45.675,158.877
C09768=1031.539,325.046,371.403,171.596,45.674,158.876
C09769=1031.531,324.798,371.437,171.592,45.673,158.875
C09770=1031.524,324.551,371.472,171.587,45.672,158.874
C09771=1031.517,324.304,371.506,171.581,45.672,158.874
C09772=1031.509,324.056,371.541,171.576,45.671,158.873
C09773=1031.502,323.808,371.576,171.571,45.671,158.872
C09774=1031.495,323.561,371.611,171.566,45.670,158.872
C09775=1031.488,323.314,371.646,171.561,45.669,158.871
C09776=1031.480,323.066,371.681,171.556,45.668,158.870
C09777=1031.473,322.819,371.716,171.551,45.668,158.870
C09778=1031.466,322.571,371.750,171.545,45.667,158.869
C09779=1031.459,322.324,371.785,171.541,45.666,158.868
C09780=1031.451,322.077,371.820,171.536,45.665,158.867
C09781=1031.443,321.829,371.855,171.530,45.665,158.867
C09782=1031.432,321.420,371.912,171.522,45.664,158.865
C09783=1031.420,321.011,371.969,171.514,45.663,158.864
C09784=1031.408,320.603,372.026,171.505,45.662,158.863
C09785=1031.397,320.194,372.084,171.497,45.661,158.862
C09786=1031.389,319.947,372.118,171.492,45.660,158.861
C09787=1031.382,319.699,372.152,171.487,45.660,158.861
C09788=1031.375,319.452,372.187,171.483,45.659,158.860
C09789=1031.368,319.204,372.221,171.477,45.659,158.859
C09790=1031.361,318.956,372.256,171.472,45.658,158.859
C09791=1031.354,318.709,372.290,171.468,45.658,158.858
C09792=1031.346,318.462,372.324,171.463,45.657,158.857
C09793=1031.340,318.214,372.360,171.458,45.656,158.857
C09794=1031.332,317.967,372.393,171.452,45.656,158.856
C09795=1031.326,317.719,372.428,171.447,45.655,158.855
C09796=1031.318,317.472,372.462,171.443,45.655,158.855
C09797=1031.311,317.224,372.496,171.438,45.654,158.854
C09798=1031.304,316.977,372.531,171.433,45.654,158.854
C09799=1031.297,316.729,372.565,171.428,45.653,158.853
C09800=1031.290,316.482,372.600,171.423,45.653,158.852
C09801=1031.283,316.234,372.634,171.418,45.652,158.851
C09802=1031.276,315.986,372.668,171.414,45.652,158.851
C09803=1031.269,315.739,372.703,171.409,45.651,158.850
C09804=1031.262,315.491,372.737,171.404,45.651,158.850
C09805=1031.256,315.243,372.771,171.400,45.650,158.849
C09806=1031.248,314.996,372.806,171.394,45.650,158.848
C09807=1031.241,314.748,372.840,171.389,45.649,158.848
C09808=1031.235,314.501,372.874,171.384,45.649,158.847
C09809=1031.228,314.254,372.908,171.380,45.648,158.846
C09810=1031.220,314.006,372.942,171.375,45.648,158.846
C09811=1031.214,313.758,372.976,171.370,45.647,158.845
C09812=1031.207,313.511,373.010,171.366,45.647,158.845
C09813=1031.200,313.263,373.045,171.361,45.647,158.844
C09814=1031.193,313.016,373.079,171.356,45.646,158.843
C09815=1031.186,312.769,373.113,171.351,45.646,158.843
C09816=1031.180,312.521,373.147,171.346,45.645,158.842
C09817=1031.172,312.273,373.181,171.341,45.645,158.842
C09818=1031.165,312.025,373.215,171.337,45.644,158.841
C09819=1031.159,311.778,373.249,171.332,45.644,158.840
C09820=1031.152,311.531,373.283,171.327,45.644,158.840
C09821=1031.145,311.283,373.316,171.323,45.643,158.839
C09822=1031.138,311.035,373.350,171.318,45.642,158.838
C09823=1031.131,310.788,373.384,171.313,45.642,158.838
C09824=1031.124,310.541,373.418,171.309,45.642,158.837
C09825=1031.117,310.293,373.451,171.303,45.642,158.837
C09826=1031.109,310.046,373.485,171.299,45.642,158.836
C09827=1031.102,309.797,373.518,171.294,45.641,158.836
C09828=1031.095,309.550,373.551,171.289,45.641,158.835
C09829=1031.088,309.303,373.585,171.285,45.641,158.834
C09830=1031.080,309.055,373.618,171.281,45.641,158.834
C09831=1031.073,308.807,373.651,171.276,45.641,158.833
C09832=1031.066,308.559,373.685,171.271,45.641,158.833
C09833=1031.060,308.312,373.719,171.267,45.640,158.832
C09834=1031.052,308.064,373.751,171.261,45.640,158.832
C09835=1031.045,307.817,373.785,171.257,45.640,158.831
C09836=1031.038,307.570,373.818,171.252,45.640,158.831
C09837=1031.031,307.321,373.852,171.247,45.639,158.830
C09838=1031.020,306.918,373.906,171.241,45.639,158.829
C09839=1031.007,306.513,373.960,171.233,45.639,158.828
C09840=1030.996,306.110,374.014,171.225,45.639,158.827
C09841=1030.985,305.706,374.069,171.218,45.638,158.827
C09842=1030.977,305.458,374.101,171.213,45.638,158.826
C09843=1030.971,305.211,374.135,171.209,45.638,158.826
C09844=1030.964,304.963,374.168,171.204,45.638,158.825
C09845=1030.957,304.716,374.201,171.200,45.638,158.824
C09846=1030.950,304.468,374.234,171.195,45.637,158.824
C09847=1030.943,304.220,374.267,171.191,45.638,158.824
C09848=1030.936,303.973,374.300,171.186,45.637,158.823
C09849=1030.929,303.725,374.333,171.182,45.637,158.822
C09850=1030.922,303.478,374.366,171.176,45.637,158.822
C09851=1030.915,303.229,374.399,171.172,45.637,158.821
C09852=1030.909,302.982,374.432,171.168,45.637,158.821
C09853=1030.901,302.734,374.465,171.164,45.637,158.820
C09854=1030.894,302.487,374.498,171.159,45.637,158.820
C09855=1030.888,302.238,374.531,171.155,45.637,158.819
C09856=1030.881,301.992,374.565,171.150,45.636,158.819
C09857=1030.873,301.744,374.597,171.146,45.636,158.818
C09858=1030.867,301.496,374.630,171.141,45.636,158.818
C09859=1030.860,301.248,374.663,171.137,45.636,158.817
C09860=1030.853,301.001,374.696,171.133,45.637,158.817
C09861=1030.846,300.753,374.729,171.128,45.636,158.816
C09862=1030.840,300.505,374.762,171.123,45.636,158.816
C09863=1030.832,300.257,374.794,171.119,45.636,158.815
C09864=1030.826,300.010,374.827,171.114,45.636,158.815
C09865=1030.819,299.761,374.860,171.110,45.636,158.814
C09866=1030.812,299.514,374.894,171.106,45.636,158.814
C09867=1030.805,299.267,374.926,171.101,45.636,158.813
C09868=1030.798,299.019,374.959,171.097,45.636,158.813
C09869=1030.792,298.771,374.992,171.092,45.636,158.812
C09870=1030.784,298.523,375.024,171.088,45.636,158.812
C09871=1030.778,298.276,375.057,171.083,45.636,158.811
C09872=1030.772,298.028,375.090,171.080,45.636,158.811
C09873=1030.764,297.780,375.122,171.075,45.636,158.811
C09874=1030.758,297.532,375.155,171.071,45.636,158.810
C09875=1030.752,297.285,375.188,171.066,45.636,158.810
C09876=1030.745,297.036,375.221,171.062,45.636,158.809
C09877=1030.738,296.789,375.253,171.058,45.636,158.809
C09878=1030.731,296.542,375.286,171.053,45.636,158.808
C09879=1030.724,296.293,375.319,171.049,45.636,158.808
C09880=1030.717,296.046,375.351,171.044,45.636,158.807
C09881=1030.711,295.798,375.384,171.041,45.636,158.807
C09882=1030.705,295.551,375.416,171.036,45.636,158.806
C09883=1030.697,295.303,375.449,171.032,45.636,158.806
C09884=1030.691,295.055,375.482,171.028,45.636,158.805
C09885=1030.685,294.807,375.514,171.023,45.636,158.805
C09886=1030.678,294.560,375.546,171.019,45.636,158.804
C09887=1030.671,294.311,375.579,171.014,45.636,158.804
C09888=1030.664,294.064,375.611,171.011,45.636,158.804
C09889=1030.658,293.816,375.643,171.006,45.636,158.803
C09890=1030.650,293.568,375.676,171.002,45.637,158.803
C09891=1030.643,293.321,375.708,170.998,45.637,158.802
C09892=1030.637,293.072,375.740,170.993,45.637,158.802
C09893=1030.630,292.825,375.772,170.989,45.637,158.801
C09894=1030.620,292.438,375.822,170.982,45.637,158.801
C09895=1030.608,292.051,375.872,170.976,45.637,158.800
C09896=1030.598,291.664,375.922,170.969,45.638,158.800
C09897=1030.587,291.278,375.973,170.963,45.638,158.799
C09898=1030.580,291.030,376.004,170.958,45.639,158.799
C09899=1030.574,290.782,376.036,170.954,45.639,158.798
C09900=1030.567,290.534,376.068,170.950,45.639,158.798
C09901=1030.560,290.286,376.100,170.946,45.639,158.797
C09902=1030.553,290.038,376.132,170.942,45.639,158.797
C09903=1030.546,289.791,376.164,170.938,45.639,158.796
C09904=1030.540,289.543,376.196,170.933,45.640,158.796
C09905=1030.533,289.295,376.228,170.929,45.640,158.796
C09906=1030.526,289.047,376.259,170.925,45.640,158.795
C09907=1030.519,288.800,376.291,170.921,45.640,158.795
C09908=1030.512,288.551,376.323,170.917,45.641,158.795
C09909=1030.506,288.303,376.355,170.913,45.641,158.794
C09910=1030.499,288.056,376.387,170.909,45.641,158.794
C09911=1030.492,287.808,376.419,170.904,45.642,158.793
C09912=1030.486,287.560,376.450,170.901,45.642,158.793
C09913=1030.479,287.312,376.482,170.897,45.642,158.793
C09914=1030.472,287.065,376.514,170.892,45.643,158.792
C09915=1030.465,286.817,376.545,170.888,45.643,158.792
C09916=1030.458,286.569,376.577,170.884,45.643,158.791
C09917=1030.452,286.321,376.609,170.880,45.643,158.791
C09918=1030.445,286.073,376.641,170.876,45.644,158.791
C09919=1030.438,285.825,376.673,170.872,45.644,158.790
C09920=1030.431,285.577,376.704,170.867,45.644,158.790
C09921=1030.424,285.329,376.735,170.863,45.645,158.790
C09922=1030.417,285.081,376.766,170.859,45.646,158.789
C09923=1030.410,284.834,376.798,170.856,45.646,158.789
C09924=1030.404,284.586,376.829,170.851,45.646,158.789
C09925=1030.397,284.338,376.861,170.847,45.646,158.788
C09926=1030.390,284.090,376.892,170.843,45.647,158.788
C09927=1030.383,283.842,376.924,170.840,45.647,158.788
C09928=1030.377,283.594,376.955,170.835,45.648,158.787
C09929=1030.370,283.346,376.986,170.831,45.648,158.787
C09930=1030.363,283.098,377.018,170.827,45.648,158.786
C09931=1030.357,282.850,377.049,170.823,45.649,158.786
C09932=1030.350,282.602,377.081,170.819,45.649,158.786
C09933=1030.342,282.355,377.112,170.815,45.650,158.786
C09934=1030.336,282.106,377.142,170.811,45.650,158.785
C09935=1030.329,281.858,377.174,170.807,45.650,158.785
C09936=1030.323,281.611,377.205,170.804,45.651,158.785
C09937=1030.316,281.363,377.237,170.799,45.651,158.784
C09938=1030.309,281.115,377.268,170.795,45.652,158.784
C09939=1030.302,280.867,377.299,170.791,45.653,158.784
C09940=1030.296,280.619,377.331,170.788,45.653,158.783
C09941=1030.289,280.370,377.362,170.783,45.653,158.783
C09942=1030.282,280.122,377.393,170.779,45.654,158.782
C09943=1030.275,279.875,377.424,170.775,45.654,158.782
C09944=1030.268,279.627,377.455,170.772,45.655,158.782
C09945=1030.262,279.380,377.486,170.767,45.655,158.781
C09946=1030.256,279.131,377.517,170.763,45.656,158.781
C09947=1030.249,278.883,377.549,170.760,45.656,158.781
C09948=1030.242,278.635,377.580,170.756,45.656,158.781
C09949=1030.236,278.387,377.611,170.752,45.657,158.780
C09950=1030.226,278.012,377.658,170.746,45.658,158.780
C09951=1030.215,277.638,377.704,170.740,45.659,158.779
C09952=1030.205,277.263,377.752,170.734,45.659,158.779
C09953=1030.195,276.888,377.798,170.728,45.660,158.778
C09954=1030.189,276.641,377.829,170.724,45.661,158.778
C09955=1030.182,276.392,377.859,170.720,45.661,158.778
C09956=1030.175,276.145,377.890,170.717,45.662,158.778
C09957=1030.168,275.896,377.921,170.713,45.662,158.777
C09958=1030.162,275.648,377.952,170.709,45.663,158.777
C09959=1030.154,275.400,377.983,170.705,45.663,158.777
C09960=1030.148,275.153,378.014,170.701,45.664,158.776
C09961=1030.142,274.905,378.044,170.697,45.665,158.776
C09962=1030.134,274.657,378.075,170.693,45.666,158.776
C09963=1030.128,274.408,378.106,170.690,45.666,158.775
C09964=1030.121,274.160,378.136,170.685,45.667,158.775
C09965=1030.115,273.913,378.167,170.681,45.668,158.775
C09966=1030.108,273.664,378.198,170.678,45.668,158.775
C09967=1030.101,273.417,378.229,170.674,45.669,158.774
C09968=1030.094,273.168,378.259,170.670,45.669,158.774
C09969=1030.088,272.921,378.289,170.667,45.670,158.774
C09970=1030.081,272.672,378.320,170.663,45.671,158.774
C09971=1030.075,272.424,378.351,170.658,45.671,158.773
C09972=1030.068,272.176,378.381,170.655,45.672,158.773
C09973=1030.062,271.928,378.412,170.651,45.673,158.773
C09974=1030.054,271.681,378.443,170.647,45.673,158.772
C09975=1030.048,271.432,378.473,170.644,45.674,158.772
C09976=1030.041,271.184,378.503,170.640,45.674,158.772
C09977=1030.035,270.936,378.534,170.637,45.675,158.772
C09978=1030.028,270.688,378.564,170.633,45.676,158.771
C09979=1030.021,270.440,378.595,170.629,45.677,158.771
C09980=1030.014,270.193,378.625,170.625,45.677,158.771
C09981=1030.008,269.944,378.656,170.621,45.678,158.771
C09982=1030.001,269.696,378.686,170.617,45.679,158.770
C09983=1029.994,269.448,378.716,170.614,45.679,158.770
C09984=1029.988,269.200,378.746,170.610,45.680,158.770
C09985=1029.981,268.952,378.776,170.606,45.681,158.770
C09986=1029.974,268.703,378.807,170.603,45.681,158.770
C09987=1029.968,268.456,378.837,170.599,45.682,158.769
C09988=1029.961,268.207,378.867,170.594,45.683,158.769
C09989=1029.955,267.960,378.897,170.591,45.683,158.769
C09990=1029.948,267.711,378.928,170.587,45.684,158.768
C09991=1029.941,267.463,378.958,170.584,45.685,158.768
C09992=1029.935,267.215,378.988,170.580,45.686,158.768
C09993=1029.927,266.967,379.018,170.576,45.687,158.768
C09994=1029.921,266.719,379.049,170.573,45.687,158.768
C09995=1029.914,266.471,379.079,170.569,45.688,158.767
C09996=1029.907,266.223,379.109,170.566,45.689,158.767
//INST
///DATE 2021/06/25 14:49
///ATTR SC,RW,RJ
////FRAME ROBOT
///GROUP1 RB1
NOP
MOVL C00000 V=800.0 PL=0
MOVL C00001 V=800.0 PL=0
MOVL C00002 V=800.0 PL=0
MOVL C00003 V=800.0 PL=0
MOVL C00004 V=800.0 PL=0
MOVL C00005 V=800.0 PL=0
MOVL C00006 V=800.0 PL=0
MOVL C00007 V=800.0 PL=0
MOVL C00008 V=800.0 PL=0
MOVL C00009 V=800.0 PL=0
MOVL C00010 V=800.0 PL=0
MOVL C00011 V=800.0 PL=0
MOVL C00012 V=800.0 PL=0
MOVL C00013 V=800.0 PL=0
MOVL C00014 V=800.0 PL=0
MOVL C00015 V=800.0 PL=0
MOVL C00016 V=800.0 PL=0
MOVL C00017 V=800.0 PL=0
MOVL C00018 V=800.0 PL=0
MOVL C00019 V=800.0 PL=0
MOVL C00020 V=800.0 PL=0
MOVL C00021 V=800.0 PL=0
MOVL C00022 V=800.0 PL=0
MOVL C00023 V=800.0 PL=0
MOVL C00024 V=800.0 PL=0
MOVL C00025 V=800.0 PL=0
MOVL C00026 V=800.0 PL=0
MOVL C00027 V=800.0 PL=0
MOVL C00028 V=800.0 PL=0
MOVL C00029 V=800.0 PL=0
MOVL C00030 V=800.0 PL=0
MOVL C00031 V=800.0 PL=0
MOVL C00032 V=800.0 PL=0
MOVL C00033 V=800.0 PL=0
MOVL C00034 V=800.0 PL=0
MOVL C00035 V=800.0 PL=0
MOVL C00036 V=800.0 PL=0
MOVL C00037 V=800.0 PL=0
MOVL C00038 V=800.0 PL=0
MOVL C00039 V=800.0 PL=0
MOVL C00040 V=800.0 PL=0
MOVL C00041 V=800.0 PL=0
MOVL C00042 V=800.0 PL=0
MOVL C00043 V=800.0 PL=0
MOVL C00044 V=800.0 PL=0
MOVL C00045 V=800.0 PL=0
MOVL C00046 V=800.0 PL=0
MOVL C00047 V=800.0 PL=0
MOVL C00048 V=800.0 PL=0
MOVL C00049 V=800.0 PL=0
MOVL C00050 V=800.0 PL=0
MOVL C00051 V=800.0 PL=0
MOVL C00052 V=800.0 PL=0
MOVL C00053 V=800.0 PL=0
MOVL C00054 V=800.0 PL=0
MOVL C00055 V=800.0 PL=0
MOVL C00056 V=800.0 PL=0
MOVL C00057 V=800.0 PL=0
MOVL C00058 V=800.0 PL=0
MOVL C00059 V=800.0 PL=0
MOVL C00060 V=800.0 PL=0
MOVL C00061 V=800.0 PL=0
MOVL C00062 V=800.0 PL=0
MOVL C00063 V=800.0 PL=0
MOVL C00064 V=800.0 PL=0
MOVL C00065 V=800.0 PL=0
MOVL C00066 V=800.0 PL=0
MOVL C00067 V=800.0 PL=0
MOVL C00068 V=800.0 PL=0
MOVL C00069 V=800.0 PL=0
MOVL C00070 V=800.0 PL=0
MOVL C00071 V=800.0 PL=0
MOVL C00072 V=800.0 PL=0
MOVL C00073 V=800.0 PL=0
MOVL C00074 V=800.0 PL=0
MOVL C00075 V=800.0 PL=0
MOVL C00076 V=800.0 PL=0
MOVL C00077 V=800.0 PL=0
MOVL C00078 V=800.0 PL=0
MOVL C00079 V=800.0 PL=0
MOVL C00080 V=800.0 PL=0
MOVL C00081 V=800.0 PL=0
MOVL C00082 V=800.0 PL=0
MOVL C00083 V=800.0 PL=0
MOVL C00084 V=800.0 PL=0
MOVL C00085 V=800.0 PL=0
MOVL C00086 V=800.0 PL=0
MOVL C00087 V=800.0 PL=0
MOVL C00088 V=800.0 PL=0
MOVL C00089 V=800.0 PL=0
MOVL C00090 V=800.0 PL=0
MOVL C00091 V=800.0 PL=0
MOVL C00092 V=800.0 PL=0
MOVL C00093 V=800.0 PL=0
MOVL C00094 V=800.0 PL=0
MOVL C00095 V=800.0 PL=0
MOVL C00096 V=800.0 PL=0
MOVL C00097 V=800.0 PL=0
MOVL C00098 V=800.0 PL=0
MOVL C00099 V=800.0 PL=0
MOVL C00100 V=800.0 PL=0
MOVL C00101 V=800.0 PL=0
MOVL C00102 V=800.0 PL=0
MOVL C00103 V=800.0 PL=0
MOVL C00104 V=800.0 PL=0
MOVL C00105 V=800.0 PL=0
MOVL C00106 V=800.0 PL=0
MOVL C00107 V=800.0 PL=0
MOVL C00108 V=800.0 PL=0
MOVL C00109 V=800.0 PL=0
MOVL C00110 V=800.0 PL=0
MOVL C00111 V=800.0 PL=0
MOVL C00112 V=800.0 PL=0
MOVL C00113 V=800.0 PL=0
MOVL C00114 V=800.0 PL=0
MOVL C00115 V=800.0 PL=0
MOVL C00116 V=800.0 PL=0
MOVL C00117 V=800.0 PL=0
MOVL C00118 V=800.0 PL=0
MOVL C00119 V=800.0 PL=0
MOVL C00120 V=800.0 PL=0
MOVL C00121 V=800.0 PL=0
MOVL C00122 V=800.0 PL=0
MOVL C00123 V=800.0 PL=0
MOVL C00124 V=800.0 PL=0
MOVL C00125 V=800.0 PL=0
MOVL C00126 V=800.0 PL=0
MOVL C00127 V=800.0 PL=0
MOVL C00128 V=800.0 PL=0
MOVL C00129 V=800.0 PL=0
MOVL C00130 V=800.0 PL=0
MOVL C00131 V=800.0 PL=0
MOVL C00132 V=800.0 PL=0
MOVL C00133 V=800.0 PL=0
MOVL C00134 V=800.0 PL=0
MOVL C00135 V=800.0 PL=0
MOVL C00136 V=800.0 PL=0
MOVL C00137 V=800.0 PL=0
MOVL C00138 V=800.0 PL=0
MOVL C00139 V=800.0 PL=0
MOVL C00140 V=800.0 PL=0
MOVL C00141 V=800.0 PL=0
MOVL C00142 V=800.0 PL=0
MOVL C00143 V=800.0 PL=0
MOVL C00144 V=800.0 PL=0
MOVL C00145 V=800.0 PL=0
MOVL C00146 V=800.0 PL=0
MOVL C00147 V=800.0 PL=0
MOVL C00148 V=800.0 PL=0
MOVL C00149 V=800.0 PL=0
MOVL C00150 V=800.0 PL=0
MOVL C00151 V=800.0 PL=0
MOVL C00152 V=800.0 PL=0
MOVL C00153 V=800.0 PL=0
MOVL C00154 V=800.0 PL=0
MOVL C00155 V=800.0 PL=0
MOVL C00156 V=800.0 PL=0
MOVL C00157 V=800.0 PL=0
MOVL C00158 V=800.0 PL=0
MOVL C00159 V=800.0 PL=0
MOVL C00160 V=800.0 PL=0
MOVL C00161 V=800.0 PL=0
MOVL C00162 V=800.0 PL=0
MOVL C00163 V=800.0 PL=0
MOVL C00164 V=800.0 PL=0
MOVL C00165 V=800.0 PL=0
MOVL C00166 V=800.0 PL=0
MOVL C00167 V=800.0 PL=0
MOVL C00168 V=800.0 PL=0
MOVL C00169 V=800.0 PL=0
MOVL C00170 V=800.0 PL=0
MOVL C00171 V=800.0 PL=0
MOVL C00172 V=800.0 PL=0
MOVL C00173 V=800.0 PL=0
MOVL C00174 V=800.0 PL=0
MOVL C00175 V=800.0 PL=0
MOVL C00176 V=800.0 PL=0
MOVL C00177 V=800.0 PL=0
MOVL C00178 V=800.0 PL=0
MOVL C00179 V=800.0 PL=0
MOVL C00180 V=800.0 PL=0
MOVL C00181 V=800.0 PL=0
MOVL C00182 V=800.0 PL=0
MOVL C00183 V=800.0 PL=0
MOVL C00184 V=800.0 PL=0
MOVL C00185 V=800.0 PL=0
MOVL C00186 V=800.0 PL=0
MOVL C00187 V=800.0 PL=0
MOVL C00188 V=800.0 PL=0
MOVL C00189 V=800.0 PL=0
MOVL C00190 V=800.0 PL=0
MOVL C00191 V=800.0 PL=0
MOVL C00192 V=800.0 PL=0
MOVL C00193 V=800.0 PL=0
MOVL C00194 V=800.0 PL=0
MOVL C00195 V=800.0 PL=0
MOVL C00196 V=800.0 PL=0
MOVL C00197 V=800.0 PL=0
MOVL C00198 V=800.0 PL=0
MOVL C00199 V=800.0 PL=0
MOVL C00200 V=800.0 PL=0
MOVL C00201 V=800.0 PL=0
MOVL C00202 V=800.0 PL=0
MOVL C00203 V=800.0 PL=0
MOVL C00204 V=800.0 PL=0
MOVL C00205 V=800.0 PL=0
MOVL C00206 V=800.0 PL=0
MOVL C00207 V=800.0 PL=0
MOVL C00208 V=800.0 PL=0
MOVL C00209 V=800.0 PL=0
MOVL C00210 V=800.0 PL=0
MOVL C00211 V=800.0 PL=0
MOVL C00212 V=800.0 PL=0
MOVL C00213 V=800.0 PL=0
MOVL C00214 V=800.0 PL=0
MOVL C00215 V=800.0 PL=0
MOVL C00216 V=800.0 PL=0
MOVL C00217 V=800.0 PL=0
MOVL C00218 V=800.0 PL=0
MOVL C00219 V=800.0 PL=0
MOVL C00220 V=800.0 PL=0
MOVL C00221 V=800.0 PL=0
MOVL C00222 V=800.0 PL=0
MOVL C00223 V=800.0 PL=0
MOVL C00224 V=800.0 PL=0
MOVL C00225 V=800.0 PL=0
MOVL C00226 V=800.0 PL=0
MOVL C00227 V=800.0 PL=0
MOVL C00228 V=800.0 PL=0
MOVL C00229 V=800.0 PL=0
MOVL C00230 V=800.0 PL=0
MOVL C00231 V=800.0 PL=0
MOVL C00232 V=800.0 PL=0
MOVL C00233 V=800.0 PL=0
MOVL C00234 V=800.0 PL=0
MOVL C00235 V=800.0 PL=0
MOVL C00236 V=800.0 PL=0
MOVL C00237 V=800.0 PL=0
MOVL C00238 V=800.0 PL=0
MOVL C00239 V=800.0 PL=0
MOVL C00240 V=800.0 PL=0
MOVL C00241 V=800.0 PL=0
MOVL C00242 V=800.0 PL=0
MOVL C00243 V=800.0 PL=0
MOVL C00244 V=800.0 PL=0
MOVL C00245 V=800.0 PL=0
MOVL C00246 V=800.0 PL=0
MOVL C00247 V=800.0 PL=0
MOVL C00248 V=800.0 PL=0
MOVL C00249 V=800.0 PL=0
MOVL C00250 V=800.0 PL=0
MOVL C00251 V=800.0 PL=0
MOVL C00252 V=800.0 PL=0
MOVL C00253 V=800.0 PL=0
MOVL C00254 V=800.0 PL=0
MOVL C00255 V=800.0 PL=0
MOVL C00256 V=800.0 PL=0
MOVL C00257 V=800.0 PL=0
MOVL C00258 V=800.0 PL=0
MOVL C00259 V=800.0 PL=0
MOVL C00260 V=800.0 PL=0
MOVL C00261 V=800.0 PL=0
MOVL C00262 V=800.0 PL=0
MOVL C00263 V=800.0 PL=0
MOVL C00264 V=800.0 PL=0
MOVL C00265 V=800.0 PL=0
MOVL C00266 V=800.0 PL=0
MOVL C00267 V=800.0 PL=0
MOVL C00268 V=800.0 PL=0
MOVL C00269 V=800.0 PL=0
MOVL C00270 V=800.0 PL=0
MOVL C00271 V=800.0 PL=0
MOVL C00272 V=800.0 PL=0
MOVL C00273 V=800.0 PL=0
MOVL C00274 V=800.0 PL=0
MOVL C00275 V=800.0 PL=0
MOVL C00276 V=800.0 PL=0
MOVL C00277 V=800.0 PL=0
MOVL C00278 V=800.0 PL=0
MOVL C00279 V=800.0 PL=0
MOVL C00280 V=800.0 PL=0
MOVL C00281 V=800.0 PL=0
MOVL C00282 V=800.0 PL=0
MOVL C00283 V=800.0 PL=0
MOVL C00284 V=800.0 PL=0
MOVL C00285 V=800.0 PL=0
MOVL C00286 V=800.0 PL=0
MOVL C00287 V=800.0 PL=0
MOVL C00288 V=800.0 PL=0
MOVL C00289 V=800.0 PL=0
MOVL C00290 V=800.0 PL=0
MOVL C00291 V=800.0 PL=0
MOVL C00292 V=800.0 PL=0
MOVL C00293 V=800.0 PL=0
MOVL C00294 V=800.0 PL=0
MOVL C00295 V=800.0 PL=0
MOVL C00296 V=800.0 PL=0
MOVL C00297 V=800.0 PL=0
MOVL C00298 V=800.0 PL=0
MOVL C00299 V=800.0 PL=0
MOVL C00300 V=800.0 PL=0
MOVL C00301 V=800.0 PL=0
MOVL C00302 V=800.0 PL=0
MOVL C00303 V=800.0 PL=0
MOVL C00304 V=800.0 PL=0
MOVL C00305 V=800.0 PL=0
MOVL C00306 V=800.0 PL=0
MOVL C00307 V=800.0 PL=0
MOVL C00308 V=800.0 PL=0
MOVL C00309 V=800.0 PL=0
MOVL C00310 V=800.0 PL=0
MOVL C00311 V=800.0 PL=0
MOVL C00312 V=800.0 PL=0
MOVL C00313 V=800.0 PL=0
MOVL C00314 V=800.0 PL=0
MOVL C00315 V=800.0 PL=0
MOVL C00316 V=800.0 PL=0
MOVL C00317 V=800.0 PL=0
MOVL C00318 V=800.0 PL=0
MOVL C00319 V=800.0 PL=0
MOVL C00320 V=800.0 PL=0
MOVL C00321 V=800.0 PL=0
MOVL C00322 V=800.0 PL=0
MOVL C00323 V=800.0 PL=0
MOVL C00324 V=800.0 PL=0
MOVL C00325 V=800.0 PL=0
MOVL C00326 V=800.0 PL=0
MOVL C00327 V=800.0 PL=0
MOVL C00328 V=800.0 PL=0
MOVL C00329 V=800.0 PL=0
MOVL C00330 V=800.0 PL=0
MOVL C00331 V=800.0 PL=0
MOVL C00332 V=800.0 PL=0
MOVL C00333 V=800.0 PL=0
MOVL C00334 V=800.0 PL=0
MOVL C00335 V=800.0 PL=0
MOVL C00336 V=800.0 PL=0
MOVL C00337 V=800.0 PL=0
MOVL C00338 V=800.0 PL=0
MOVL C00339 V=800.0 PL=0
MOVL C00340 V=800.0 PL=0
MOVL C00341 V=800.0 PL=0
MOVL C00342 V=800.0 PL=0
MOVL C00343 V=800.0 PL=0
MOVL C00344 V=800.0 PL=0
MOVL C00345 V=800.0 PL=0
MOVL C00346 V=800.0 PL=0
MOVL C00347 V=800.0 PL=0
MOVL C00348 V=800.0 PL=0
MOVL C00349 V=800.0 PL=0
MOVL C00350 V=800.0 PL=0
MOVL C00351 V=800.0 PL=0
MOVL C00352 V=800.0 PL=0
MOVL C00353 V=800.0 PL=0
MOVL C00354 V=800.0 PL=0
MOVL C00355 V=800.0 PL=0
MOVL C00356 V=800.0 PL=0
MOVL C00357 V=800.0 PL=0
MOVL C00358 V=800.0 PL=0
MOVL C00359 V=800.0 PL=0
MOVL C00360 V=800.0 PL=0
MOVL C00361 V=800.0 PL=0
MOVL C00362 V=800.0 PL=0
MOVL C00363 V=800.0 PL=0
MOVL C00364 V=800.0 PL=0
MOVL C00365 V=800.0 PL=0
MOVL C00366 V=800.0 PL=0
MOVL C00367 V=800.0 PL=0
MOVL C00368 V=800.0 PL=0
MOVL C00369 V=800.0 PL=0
MOVL C00370 V=800.0 PL=0
MOVL C00371 V=800.0 PL=0
MOVL C00372 V=800.0 PL=0
MOVL C00373 V=800.0 PL=0
MOVL C00374 V=800.0 PL=0
MOVL C00375 V=800.0 PL=0
MOVL C00376 V=800.0 PL=0
MOVL C00377 V=800.0 PL=0
MOVL C00378 V=800.0 PL=0
MOVL C00379 V=800.0 PL=0
MOVL C00380 V=800.0 PL=0
MOVL C00381 V=800.0 PL=0
MOVL C00382 V=800.0 PL=0
MOVL C00383 V=800.0 PL=0
MOVL C00384 V=800.0 PL=0
MOVL C00385 V=800.0 PL=0
MOVL C00386 V=800.0 PL=0
MOVL C00387 V=800.0 PL=0
MOVL C00388 V=800.0 PL=0
MOVL C00389 V=800.0 PL=0
MOVL C00390 V=800.0 PL=0
MOVL C00391 V=800.0 PL=0
MOVL C00392 V=800.0 PL=0
MOVL C00393 V=800.0 PL=0
MOVL C00394 V=800.0 PL=0
MOVL C00395 V=800.0 PL=0
MOVL C00396 V=800.0 PL=0
MOVL C00397 V=800.0 PL=0
MOVL C00398 V=800.0 PL=0
MOVL C00399 V=800.0 PL=0
MOVL C00400 V=800.0 PL=0
MOVL C00401 V=800.0 PL=0
MOVL C00402 V=800.0 PL=0
MOVL C00403 V=800.0 PL=0
MOVL C00404 V=800.0 PL=0
MOVL C00405 V=800.0 PL=0
MOVL C00406 V=800.0 PL=0
MOVL C00407 V=800.0 PL=0
MOVL C00408 V=800.0 PL=0
MOVL C00409 V=800.0 PL=0
MOVL C00410 V=800.0 PL=0
MOVL C00411 V=800.0 PL=0
MOVL C00412 V=800.0 PL=0
MOVL C00413 V=800.0 PL=0
MOVL C00414 V=800.0 PL=0
MOVL C00415 V=800.0 PL=0
MOVL C00416 V=800.0 PL=0
MOVL C00417 V=800.0 PL=0
MOVL C00418 V=800.0 PL=0
MOVL C00419 V=800.0 PL=0
MOVL C00420 V=800.0 PL=0
MOVL C00421 V=800.0 PL=0
MOVL C00422 V=800.0 PL=0
MOVL C00423 V=800.0 PL=0
MOVL C00424 V=800.0 PL=0
MOVL C00425 V=800.0 PL=0
MOVL C00426 V=800.0 PL=0
MOVL C00427 V=800.0 PL=0
MOVL C00428 V=800.0 PL=0
MOVL C00429 V=800.0 PL=0
MOVL C00430 V=800.0 PL=0
MOVL C00431 V=800.0 PL=0
MOVL C00432 V=800.0 PL=0
MOVL C00433 V=800.0 PL=0
MOVL C00434 V=800.0 PL=0
MOVL C00435 V=800.0 PL=0
MOVL C00436 V=800.0 PL=0
MOVL C00437 V=800.0 PL=0
MOVL C00438 V=800.0 PL=0
MOVL C00439 V=800.0 PL=0
MOVL C00440 V=800.0 PL=0
MOVL C00441 V=800.0 PL=0
MOVL C00442 V=800.0 PL=0
MOVL C00443 V=800.0 PL=0
MOVL C00444 V=800.0 PL=0
MOVL C00445 V=800.0 PL=0
MOVL C00446 V=800.0 PL=0
MOVL C00447 V=800.0 PL=0
MOVL C00448 V=800.0 PL=0
MOVL C00449 V=800.0 PL=0
MOVL C00450 V=800.0 PL=0
MOVL C00451 V=800.0 PL=0
MOVL C00452 V=800.0 PL=0
MOVL C00453 V=800.0 PL=0
MOVL C00454 V=800.0 PL=0
MOVL C00455 V=800.0 PL=0
MOVL C00456 V=800.0 PL=0
MOVL C00457 V=800.0 PL=0
MOVL C00458 V=800.0 PL=0
MOVL C00459 V=800.0 PL=0
MOVL C00460 V=800.0 PL=0
MOVL C00461 V=800.0 PL=0
MOVL C00462 V=800.0 PL=0
MOVL C00463 V=800.0 PL=0
MOVL C00464 V=800.0 PL=0
MOVL C00465 V=800.0 PL=0
MOVL C00466 V=800.0 PL=0
MOVL C00467 V=800.0 PL=0
MOVL C00468 V=800.0 PL=0
MOVL C00469 V=800.0 PL=0
MOVL C00470 V=800.0 PL=0
MOVL C00471 V=800.0 PL=0
MOVL C00472 V=800.0 PL=0
MOVL C00473 V=800.0 PL=0
MOVL C00474 V=800.0 PL=0
MOVL C00475 V=800.0 PL=0
MOVL C00476 V=800.0 PL=0
MOVL C00477 V=800.0 PL=0
MOVL C00478 V=800.0 PL=0
MOVL C00479 V=800.0 PL=0
MOVL C00480 V=800.0 PL=0
MOVL C00481 V=800.0 PL=0
MOVL C00482 V=800.0 PL=0
MOVL C00483 V=800.0 PL=0
MOVL C00484 V=800.0 PL=0
MOVL C00485 V=800.0 PL=0
MOVL C00486 V=800.0 PL=0
MOVL C00487 V=800.0 PL=0
MOVL C00488 V=800.0 PL=0
MOVL C00489 V=800.0 PL=0
MOVL C00490 V=800.0 PL=0
MOVL C00491 V=800.0 PL=0
MOVL C00492 V=800.0 PL=0
MOVL C00493 V=800.0 PL=0
MOVL C00494 V=800.0 PL=0
MOVL C00495 V=800.0 PL=0
MOVL C00496 V=800.0 PL=0
MOVL C00497 V=800.0 PL=0
MOVL C00498 V=800.0 PL=0
MOVL C00499 V=800.0 PL=0
MOVL C00500 V=800.0 PL=0
MOVL C00501 V=800.0 PL=0
MOVL C00502 V=800.0 PL=0
MOVL C00503 V=800.0 PL=0
MOVL C00504 V=800.0 PL=0
MOVL C00505 V=800.0 PL=0
MOVL C00506 V=800.0 PL=0
MOVL C00507 V=800.0 PL=0
MOVL C00508 V=800.0 PL=0
MOVL C00509 V=800.0 PL=0
MOVL C00510 V=800.0 PL=0
MOVL C00511 V=800.0 PL=0
MOVL C00512 V=800.0 PL=0
MOVL C00513 V=800.0 PL=0
MOVL C00514 V=800.0 PL=0
MOVL C00515 V=800.0 PL=0
MOVL C00516 V=800.0 PL=0
MOVL C00517 V=800.0 PL=0
MOVL C00518 V=800.0 PL=0
MOVL C00519 V=800.0 PL=0
MOVL C00520 V=800.0 PL=0
MOVL C00521 V=800.0 PL=0
MOVL C00522 V=800.0 PL=0
MOVL C00523 V=800.0 PL=0
MOVL C00524 V=800.0 PL=0
MOVL C00525 V=800.0 PL=0
MOVL C00526 V=800.0 PL=0
MOVL C00527 V=800.0 PL=0
MOVL C00528 V=800.0 PL=0
MOVL C00529 V=800.0 PL=0
MOVL C00530 V=800.0 PL=0
MOVL C00531 V=800.0 PL=0
MOVL C00532 V=800.0 PL=0
MOVL C00533 V=800.0 PL=0
MOVL C00534 V=800.0 PL=0
MOVL C00535 V=800.0 PL=0
MOVL C00536 V=800.0 PL=0
MOVL C00537 V=800.0 PL=0
MOVL C00538 V=800.0 PL=0
MOVL C00539 V=800.0 PL=0
MOVL C00540 V=800.0 PL=0
MOVL C00541 V=800.0 PL=0
MOVL C00542 V=800.0 PL=0
MOVL C00543 V=800.0 PL=0
MOVL C00544 V=800.0 PL=0
MOVL C00545 V=800.0 PL=0
MOVL C00546 V=800.0 PL=0
MOVL C00547 V=800.0 PL=0
MOVL C00548 V=800.0 PL=0
MOVL C00549 V=800.0 PL=0
MOVL C00550 V=800.0 PL=0
MOVL C00551 V=800.0 PL=0
MOVL C00552 V=800.0 PL=0
MOVL C00553 V=800.0 PL=0
MOVL C00554 V=800.0 PL=0
MOVL C00555 V=800.0 PL=0
MOVL C00556 V=800.0 PL=0
MOVL C00557 V=800.0 PL=0
MOVL C00558 V=800.0 PL=0
MOVL C00559 V=800.0 PL=0
MOVL C00560 V=800.0 PL=0
MOVL C00561 V=800.0 PL=0
MOVL C00562 V=800.0 PL=0
MOVL C00563 V=800.0 PL=0
MOVL C00564 V=800.0 PL=0
MOVL C00565 V=800.0 PL=0
MOVL C00566 V=800.0 PL=0
MOVL C00567 V=800.0 PL=0
MOVL C00568 V=800.0 PL=0
MOVL C00569 V=800.0 PL=0
MOVL C00570 V=800.0 PL=0
MOVL C00571 V=800.0 PL=0
MOVL C00572 V=800.0 PL=0
MOVL C00573 V=800.0 PL=0
MOVL C00574 V=800.0 PL=0
MOVL C00575 V=800.0 PL=0
MOVL C00576 V=800.0 PL=0
MOVL C00577 V=800.0 PL=0
MOVL C00578 V=800.0 PL=0
MOVL C00579 V=800.0 PL=0
MOVL C00580 V=800.0 PL=0
MOVL C00581 V=800.0 PL=0
MOVL C00582 V=800.0 PL=0
MOVL C00583 V=800.0 PL=0
MOVL C00584 V=800.0 PL=0
MOVL C00585 V=800.0 PL=0
MOVL C00586 V=800.0 PL=0
MOVL C00587 V=800.0 PL=0
MOVL C00588 V=800.0 PL=0
MOVL C00589 V=800.0 PL=0
MOVL C00590 V=800.0 PL=0
MOVL C00591 V=800.0 PL=0
MOVL C00592 V=800.0 PL=0
MOVL C00593 V=800.0 PL=0
MOVL C00594 V=800.0 PL=0
MOVL C00595 V=800.0 PL=0
MOVL C00596 V=800.0 PL=0
MOVL C00597 V=800.0 PL=0
MOVL C00598 V=800.0 PL=0
MOVL C00599 V=800.0 PL=0
MOVL C00600 V=800.0 PL=0
MOVL C00601 V=800.0 PL=0
MOVL C00602 V=800.0 PL=0
MOVL C00603 V=800.0 PL=0
MOVL C00604 V=800.0 PL=0
MOVL C00605 V=800.0 PL=0
MOVL C00606 V=800.0 PL=0
MOVL C00607 V=800.0 PL=0
MOVL C00608 V=800.0 PL=0
MOVL C00609 V=800.0 PL=0
MOVL C00610 V=800.0 PL=0
MOVL C00611 V=800.0 PL=0
MOVL C00612 V=800.0 PL=0
MOVL C00613 V=800.0 PL=0
MOVL C00614 V=800.0 PL=0
MOVL C00615 V=800.0 PL=0
MOVL C00616 V=800.0 PL=0
MOVL C00617 V=800.0 PL=0
MOVL C00618 V=800.0 PL=0
MOVL C00619 V=800.0 PL=0
MOVL C00620 V=800.0 PL=0
MOVL C00621 V=800.0 PL=0
MOVL C00622 V=800.0 PL=0
MOVL C00623 V=800.0 PL=0
MOVL C00624 V=800.0 PL=0
MOVL C00625 V=800.0 PL=0
MOVL C00626 V=800.0 PL=0
MOVL C00627 V=800.0 PL=0
MOVL C00628 V=800.0 PL=0
MOVL C00629 V=800.0 PL=0
MOVL C00630 V=800.0 PL=0
MOVL C00631 V=800.0 PL=0
MOVL C00632 V=800.0 PL=0
MOVL C00633 V=800.0 PL=0
MOVL C00634 V=800.0 PL=0
MOVL C00635 V=800.0 PL=0
MOVL C00636 V=800.0 PL=0
MOVL C00637 V=800.0 PL=0
MOVL C00638 V=800.0 PL=0
MOVL C00639 V=800.0 PL=0
MOVL C00640 V=800.0 PL=0
MOVL C00641 V=800.0 PL=0
MOVL C00642 V=800.0 PL=0
MOVL C00643 V=800.0 PL=0
MOVL C00644 V=800.0 PL=0
MOVL C00645 V=800.0 PL=0
MOVL C00646 V=800.0 PL=0
MOVL C00647 V=800.0 PL=0
MOVL C00648 V=800.0 PL=0
MOVL C00649 V=800.0 PL=0
MOVL C00650 V=800.0 PL=0
MOVL C00651 V=800.0 PL=0
MOVL C00652 V=800.0 PL=0
MOVL C00653 V=800.0 PL=0
MOVL C00654 V=800.0 PL=0
MOVL C00655 V=800.0 PL=0
MOVL C00656 V=800.0 PL=0
MOVL C00657 V=800.0 PL=0
MOVL C00658 V=800.0 PL=0
MOVL C00659 V=800.0 PL=0
MOVL C00660 V=800.0 PL=0
MOVL C00661 V=800.0 PL=0
MOVL C00662 V=800.0 PL=0
MOVL C00663 V=800.0 PL=0
MOVL C00664 V=800.0 PL=0
MOVL C00665 V=800.0 PL=0
MOVL C00666 V=800.0 PL=0
MOVL C00667 V=800.0 PL=0
MOVL C00668 V=800.0 PL=0
MOVL C00669 V=800.0 PL=0
MOVL C00670 V=800.0 PL=0
MOVL C00671 V=800.0 PL=0
MOVL C00672 V=800.0 PL=0
MOVL C00673 V=800.0 PL=0
MOVL C00674 V=800.0 PL=0
MOVL C00675 V=800.0 PL=0
MOVL C00676 V=800.0 PL=0
MOVL C00677 V=800.0 PL=0
MOVL C00678 V=800.0 PL=0
MOVL C00679 V=800.0 PL=0
MOVL C00680 V=800.0 PL=0
MOVL C00681 V=800.0 PL=0
MOVL C00682 V=800.0 PL=0
MOVL C00683 V=800.0 PL=0
MOVL C00684 V=800.0 PL=0
MOVL C00685 V=800.0 PL=0
MOVL C00686 V=800.0 PL=0
MOVL C00687 V=800.0 PL=0
MOVL C00688 V=800.0 PL=0
MOVL C00689 V=800.0 PL=0
MOVL C00690 V=800.0 PL=0
MOVL C00691 V=800.0 PL=0
MOVL C00692 V=800.0 PL=0
MOVL C00693 V=800.0 PL=0
MOVL C00694 V=800.0 PL=0
MOVL C00695 V=800.0 PL=0
MOVL C00696 V=800.0 PL=0
MOVL C00697 V=800.0 PL=0
MOVL C00698 V=800.0 PL=0
MOVL C00699 V=800.0 PL=0
MOVL C00700 V=800.0 PL=0
MOVL C00701 V=800.0 PL=0
MOVL C00702 V=800.0 PL=0
MOVL C00703 V=800.0 PL=0
MOVL C00704 V=800.0 PL=0
MOVL C00705 V=800.0 PL=0
MOVL C00706 V=800.0 PL=0
MOVL C00707 V=800.0 PL=0
MOVL C00708 V=800.0 PL=0
MOVL C00709 V=800.0 PL=0
MOVL C00710 V=800.0 PL=0
MOVL C00711 V=800.0 PL=0
MOVL C00712 V=800.0 PL=0
MOVL C00713 V=800.0 PL=0
MOVL C00714 V=800.0 PL=0
MOVL C00715 V=800.0 PL=0
MOVL C00716 V=800.0 PL=0
MOVL C00717 V=800.0 PL=0
MOVL C00718 V=800.0 PL=0
MOVL C00719 V=800.0 PL=0
MOVL C00720 V=800.0 PL=0
MOVL C00721 V=800.0 PL=0
MOVL C00722 V=800.0 PL=0
MOVL C00723 V=800.0 PL=0
MOVL C00724 V=800.0 PL=0
MOVL C00725 V=800.0 PL=0
MOVL C00726 V=800.0 PL=0
MOVL C00727 V=800.0 PL=0
MOVL C00728 V=800.0 PL=0
MOVL C00729 V=800.0 PL=0
MOVL C00730 V=800.0 PL=0
MOVL C00731 V=800.0 PL=0
MOVL C00732 V=800.0 PL=0
MOVL C00733 V=800.0 PL=0
MOVL C00734 V=800.0 PL=0
MOVL C00735 V=800.0 PL=0
MOVL C00736 V=800.0 PL=0
MOVL C00737 V=800.0 PL=0
MOVL C00738 V=800.0 PL=0
MOVL C00739 V=800.0 PL=0
MOVL C00740 V=800.0 PL=0
MOVL C00741 V=800.0 PL=0
MOVL C00742 V=800.0 PL=0
MOVL C00743 V=800.0 PL=0
MOVL C00744 V=800.0 PL=0
MOVL C00745 V=800.0 PL=0
MOVL C00746 V=800.0 PL=0
MOVL C00747 V=800.0 PL=0
MOVL C00748 V=800.0 PL=0
MOVL C00749 V=800.0 PL=0
MOVL C00750 V=800.0 PL=0
MOVL C00751 V=800.0 PL=0
MOVL C00752 V=800.0 PL=0
MOVL C00753 V=800.0 PL=0
MOVL C00754 V=800.0 PL=0
MOVL C00755 V=800.0 PL=0
MOVL C00756 V=800.0 PL=0
MOVL C00757 V=800.0 PL=0
MOVL C00758 V=800.0 PL=0
MOVL C00759 V=800.0 PL=0
MOVL C00760 V=800.0 PL=0
MOVL C00761 V=800.0 PL=0
MOVL C00762 V=800.0 PL=0
MOVL C00763 V=800.0 PL=0
MOVL C00764 V=800.0 PL=0
MOVL C00765 V=800.0 PL=0
MOVL C00766 V=800.0 PL=0
MOVL C00767 V=800.0 PL=0
MOVL C00768 V=800.0 PL=0
MOVL C00769 V=800.0 PL=0
MOVL C00770 V=800.0 PL=0
MOVL C00771 V=800.0 PL=0
MOVL C00772 V=800.0 PL=0
MOVL C00773 V=800.0 PL=0
MOVL C00774 V=800.0 PL=0
MOVL C00775 V=800.0 PL=0
MOVL C00776 V=800.0 PL=0
MOVL C00777 V=800.0 PL=0
MOVL C00778 V=800.0 PL=0
MOVL C00779 V=800.0 PL=0
MOVL C00780 V=800.0 PL=0
MOVL C00781 V=800.0 PL=0
MOVL C00782 V=800.0 PL=0
MOVL C00783 V=800.0 PL=0
MOVL C00784 V=800.0 PL=0
MOVL C00785 V=800.0 PL=0
MOVL C00786 V=800.0 PL=0
MOVL C00787 V=800.0 PL=0
MOVL C00788 V=800.0 PL=0
MOVL C00789 V=800.0 PL=0
MOVL C00790 V=800.0 PL=0
MOVL C00791 V=800.0 PL=0
MOVL C00792 V=800.0 PL=0
MOVL C00793 V=800.0 PL=0
MOVL C00794 V=800.0 PL=0
MOVL C00795 V=800.0 PL=0
MOVL C00796 V=800.0 PL=0
MOVL C00797 V=800.0 PL=0
MOVL C00798 V=800.0 PL=0
MOVL C00799 V=800.0 PL=0
MOVL C00800 V=800.0 PL=0
MOVL C00801 V=800.0 PL=0
MOVL C00802 V=800.0 PL=0
MOVL C00803 V=800.0 PL=0
MOVL C00804 V=800.0 PL=0
MOVL C00805 V=800.0 PL=0
MOVL C00806 V=800.0 PL=0
MOVL C00807 V=800.0 PL=0
MOVL C00808 V=800.0 PL=0
MOVL C00809 V=800.0 PL=0
MOVL C00810 V=800.0 PL=0
MOVL C00811 V=800.0 PL=0
MOVL C00812 V=800.0 PL=0
MOVL C00813 V=800.0 PL=0
MOVL C00814 V=800.0 PL=0
MOVL C00815 V=800.0 PL=0
MOVL C00816 V=800.0 PL=0
MOVL C00817 V=800.0 PL=0
MOVL C00818 V=800.0 PL=0
MOVL C00819 V=800.0 PL=0
MOVL C00820 V=800.0 PL=0
MOVL C00821 V=800.0 PL=0
MOVL C00822 V=800.0 PL=0
MOVL C00823 V=800.0 PL=0
MOVL C00824 V=800.0 PL=0
MOVL C00825 V=800.0 PL=0
MOVL C00826 V=800.0 PL=0
MOVL C00827 V=800.0 PL=0
MOVL C00828 V=800.0 PL=0
MOVL C00829 V=800.0 PL=0
MOVL C00830 V=800.0 PL=0
MOVL C00831 V=800.0 PL=0
MOVL C00832 V=800.0 PL=0
MOVL C00833 V=800.0 PL=0
MOVL C00834 V=800.0 PL=0
MOVL C00835 V=800.0 PL=0
MOVL C00836 V=800.0 PL=0
MOVL C00837 V=800.0 PL=0
MOVL C00838 V=800.0 PL=0
MOVL C00839 V=800.0 PL=0
MOVL C00840 V=800.0 PL=0
MOVL C00841 V=800.0 PL=0
MOVL C00842 V=800.0 PL=0
MOVL C00843 V=800.0 PL=0
MOVL C00844 V=800.0 PL=0
MOVL C00845 V=800.0 PL=0
MOVL C00846 V=800.0 PL=0
MOVL C00847 V=800.0 PL=0
MOVL C00848 V=800.0 PL=0
MOVL C00849 V=800.0 PL=0
MOVL C00850 V=800.0 PL=0
MOVL C00851 V=800.0 PL=0
MOVL C00852 V=800.0 PL=0
MOVL C00853 V=800.0 PL=0
MOVL C00854 V=800.0 PL=0
MOVL C00855 V=800.0 PL=0
MOVL C00856 V=800.0 PL=0
MOVL C00857 V=800.0 PL=0
MOVL C00858 V=800.0 PL=0
MOVL C00859 V=800.0 PL=0
MOVL C00860 V=800.0 PL=0
MOVL C00861 V=800.0 PL=0
MOVL C00862 V=800.0 PL=0
MOVL C00863 V=800.0 PL=0
MOVL C00864 V=800.0 PL=0
MOVL C00865 V=800.0 PL=0
MOVL C00866 V=800.0 PL=0
MOVL C00867 V=800.0 PL=0
MOVL C00868 V=800.0 PL=0
MOVL C00869 V=800.0 PL=0
MOVL C00870 V=800.0 PL=0
MOVL C00871 V=800.0 PL=0
MOVL C00872 V=800.0 PL=0
MOVL C00873 V=800.0 PL=0
MOVL C00874 V=800.0 PL=0
MOVL C00875 V=800.0 PL=0
MOVL C00876 V=800.0 PL=0
MOVL C00877 V=800.0 PL=0
MOVL C00878 V=800.0 PL=0
MOVL C00879 V=800.0 PL=0
MOVL C00880 V=800.0 PL=0
MOVL C00881 V=800.0 PL=0
MOVL C00882 V=800.0 PL=0
MOVL C00883 V=800.0 PL=0
MOVL C00884 V=800.0 PL=0
MOVL C00885 V=800.0 PL=0
MOVL C00886 V=800.0 PL=0
MOVL C00887 V=800.0 PL=0
MOVL C00888 V=800.0 PL=0
MOVL C00889 V=800.0 PL=0
MOVL C00890 V=800.0 PL=0
MOVL C00891 V=800.0 PL=0
MOVL C00892 V=800.0 PL=0
MOVL C00893 V=800.0 PL=0
MOVL C00894 V=800.0 PL=0
MOVL C00895 V=800.0 PL=0
MOVL C00896 V=800.0 PL=0
MOVL C00897 V=800.0 PL=0
MOVL C00898 V=800.0 PL=0
MOVL C00899 V=800.0 PL=0
MOVL C00900 V=800.0 PL=0
MOVL C00901 V=800.0 PL=0
MOVL C00902 V=800.0 PL=0
MOVL C00903 V=800.0 PL=0
MOVL C00904 V=800.0 PL=0
MOVL C00905 V=800.0 PL=0
MOVL C00906 V=800.0 PL=0
MOVL C00907 V=800.0 PL=0
MOVL C00908 V=800.0 PL=0
MOVL C00909 V=800.0 PL=0
MOVL C00910 V=800.0 PL=0
MOVL C00911 V=800.0 PL=0
MOVL C00912 V=800.0 PL=0
MOVL C00913 V=800.0 PL=0
MOVL C00914 V=800.0 PL=0
MOVL C00915 V=800.0 PL=0
MOVL C00916 V=800.0 PL=0
MOVL C00917 V=800.0 PL=0
MOVL C00918 V=800.0 PL=0
MOVL C00919 V=800.0 PL=0
MOVL C00920 V=800.0 PL=0
MOVL C00921 V=800.0 PL=0
MOVL C00922 V=800.0 PL=0
MOVL C00923 V=800.0 PL=0
MOVL C00924 V=800.0 PL=0
MOVL C00925 V=800.0 PL=0
MOVL C00926 V=800.0 PL=0
MOVL C00927 V=800.0 PL=0
MOVL C00928 V=800.0 PL=0
MOVL C00929 V=800.0 PL=0
MOVL C00930 V=800.0 PL=0
MOVL C00931 V=800.0 PL=0
MOVL C00932 V=800.0 PL=0
MOVL C00933 V=800.0 PL=0
MOVL C00934 V=800.0 PL=0
MOVL C00935 V=800.0 PL=0
MOVL C00936 V=800.0 PL=0
MOVL C00937 V=800.0 PL=0
MOVL C00938 V=800.0 PL=0
MOVL C00939 V=800.0 PL=0
MOVL C00940 V=800.0 PL=0
MOVL C00941 V=800.0 PL=0
MOVL C00942 V=800.0 PL=0
MOVL C00943 V=800.0 PL=0
MOVL C00944 V=800.0 PL=0
MOVL C00945 V=800.0 PL=0
MOVL C00946 V=800.0 PL=0
MOVL C00947 V=800.0 PL=0
MOVL C00948 V=800.0 PL=0
MOVL C00949 V=800.0 PL=0
MOVL C00950 V=800.0 PL=0
MOVL C00951 V=800.0 PL=0
MOVL C00952 V=800.0 PL=0
MOVL C00953 V=800.0 PL=0
MOVL C00954 V=800.0 PL=0
MOVL C00955 V=800.0 PL=0
MOVL C00956 V=800.0 PL=0
MOVL C00957 V=800.0 PL=0
MOVL C00958 V=800.0 PL=0
MOVL C00959 V=800.0 PL=0
MOVL C00960 V=800.0 PL=0
MOVL C00961 V=800.0 PL=0
MOVL C00962 V=800.0 PL=0
MOVL C00963 V=800.0 PL=0
MOVL C00964 V=800.0 PL=0
MOVL C00965 V=800.0 PL=0
MOVL C00966 V=800.0 PL=0
MOVL C00967 V=800.0 PL=0
MOVL C00968 V=800.0 PL=0
MOVL C00969 V=800.0 PL=0
MOVL C00970 V=800.0 PL=0
MOVL C00971 V=800.0 PL=0
MOVL C00972 V=800.0 PL=0
MOVL C00973 V=800.0 PL=0
MOVL C00974 V=800.0 PL=0
MOVL C00975 V=800.0 PL=0
MOVL C00976 V=800.0 PL=0
MOVL C00977 V=800.0 PL=0
MOVL C00978 V=800.0 PL=0
MOVL C00979 V=800.0 PL=0
MOVL C00980 V=800.0 PL=0
MOVL C00981 V=800.0 PL=0
MOVL C00982 V=800.0 PL=0
MOVL C00983 V=800.0 PL=0
MOVL C00984 V=800.0 PL=0
MOVL C00985 V=800.0 PL=0
MOVL C00986 V=800.0 PL=0
MOVL C00987 V=800.0 PL=0
MOVL C00988 V=800.0 PL=0
MOVL C00989 V=800.0 PL=0
MOVL C00990 V=800.0 PL=0
MOVL C00991 V=800.0 PL=0
MOVL C00992 V=800.0 PL=0
MOVL C00993 V=800.0 PL=0
MOVL C00994 V=800.0 PL=0
MOVL C00995 V=800.0 PL=0
MOVL C00996 V=800.0 PL=0
MOVL C00997 V=800.0 PL=0
MOVL C00998 V=800.0 PL=0
MOVL C00999 V=800.0 PL=0
MOVL C01000 V=800.0 PL=0
MOVL C01001 V=800.0 PL=0
MOVL C01002 V=800.0 PL=0
MOVL C01003 V=800.0 PL=0
MOVL C01004 V=800.0 PL=0
MOVL C01005 V=800.0 PL=0
MOVL C01006 V=800.0 PL=0
MOVL C01007 V=800.0 PL=0
MOVL C01008 V=800.0 PL=0
MOVL C01009 V=800.0 PL=0
MOVL C01010 V=800.0 PL=0
MOVL C01011 V=800.0 PL=0
MOVL C01012 V=800.0 PL=0
MOVL C01013 V=800.0 PL=0
MOVL C01014 V=800.0 PL=0
MOVL C01015 V=800.0 PL=0
MOVL C01016 V=800.0 PL=0
MOVL C01017 V=800.0 PL=0
MOVL C01018 V=800.0 PL=0
MOVL C01019 V=800.0 PL=0
MOVL C01020 V=800.0 PL=0
MOVL C01021 V=800.0 PL=0
MOVL C01022 V=800.0 PL=0
MOVL C01023 V=800.0 PL=0
MOVL C01024 V=800.0 PL=0
MOVL C01025 V=800.0 PL=0
MOVL C01026 V=800.0 PL=0
MOVL C01027 V=800.0 PL=0
MOVL C01028 V=800.0 PL=0
MOVL C01029 V=800.0 PL=0
MOVL C01030 V=800.0 PL=0
MOVL C01031 V=800.0 PL=0
MOVL C01032 V=800.0 PL=0
MOVL C01033 V=800.0 PL=0
MOVL C01034 V=800.0 PL=0
MOVL C01035 V=800.0 PL=0
MOVL C01036 V=800.0 PL=0
MOVL C01037 V=800.0 PL=0
MOVL C01038 V=800.0 PL=0
MOVL C01039 V=800.0 PL=0
MOVL C01040 V=800.0 PL=0
MOVL C01041 V=800.0 PL=0
MOVL C01042 V=800.0 PL=0
MOVL C01043 V=800.0 PL=0
MOVL C01044 V=800.0 PL=0
MOVL C01045 V=800.0 PL=0
MOVL C01046 V=800.0 PL=0
MOVL C01047 V=800.0 PL=0
MOVL C01048 V=800.0 PL=0
MOVL C01049 V=800.0 PL=0
MOVL C01050 V=800.0 PL=0
MOVL C01051 V=800.0 PL=0
MOVL C01052 V=800.0 PL=0
MOVL C01053 V=800.0 PL=0
MOVL C01054 V=800.0 PL=0
MOVL C01055 V=800.0 PL=0
MOVL C01056 V=800.0 PL=0
MOVL C01057 V=800.0 PL=0
MOVL C01058 V=800.0 PL=0
MOVL C01059 V=800.0 PL=0
MOVL C01060 V=800.0 PL=0
MOVL C01061 V=800.0 PL=0
MOVL C01062 V=800.0 PL=0
MOVL C01063 V=800.0 PL=0
MOVL C01064 V=800.0 PL=0
MOVL C01065 V=800.0 PL=0
MOVL C01066 V=800.0 PL=0
MOVL C01067 V=800.0 PL=0
MOVL C01068 V=800.0 PL=0
MOVL C01069 V=800.0 PL=0
MOVL C01070 V=800.0 PL=0
MOVL C01071 V=800.0 PL=0
MOVL C01072 V=800.0 PL=0
MOVL C01073 V=800.0 PL=0
MOVL C01074 V=800.0 PL=0
MOVL C01075 V=800.0 PL=0
MOVL C01076 V=800.0 PL=0
MOVL C01077 V=800.0 PL=0
MOVL C01078 V=800.0 PL=0
MOVL C01079 V=800.0 PL=0
MOVL C01080 V=800.0 PL=0
MOVL C01081 V=800.0 PL=0
MOVL C01082 V=800.0 PL=0
MOVL C01083 V=800.0 PL=0
MOVL C01084 V=800.0 PL=0
MOVL C01085 V=800.0 PL=0
MOVL C01086 V=800.0 PL=0
MOVL C01087 V=800.0 PL=0
MOVL C01088 V=800.0 PL=0
MOVL C01089 V=800.0 PL=0
MOVL C01090 V=800.0 PL=0
MOVL C01091 V=800.0 PL=0
MOVL C01092 V=800.0 PL=0
MOVL C01093 V=800.0 PL=0
MOVL C01094 V=800.0 PL=0
MOVL C01095 V=800.0 PL=0
MOVL C01096 V=800.0 PL=0
MOVL C01097 V=800.0 PL=0
MOVL C01098 V=800.0 PL=0
MOVL C01099 V=800.0 PL=0
MOVL C01100 V=800.0 PL=0
MOVL C01101 V=800.0 PL=0
MOVL C01102 V=800.0 PL=0
MOVL C01103 V=800.0 PL=0
MOVL C01104 V=800.0 PL=0
MOVL C01105 V=800.0 PL=0
MOVL C01106 V=800.0 PL=0
MOVL C01107 V=800.0 PL=0
MOVL C01108 V=800.0 PL=0
MOVL C01109 V=800.0 PL=0
MOVL C01110 V=800.0 PL=0
MOVL C01111 V=800.0 PL=0
MOVL C01112 V=800.0 PL=0
MOVL C01113 V=800.0 PL=0
MOVL C01114 V=800.0 PL=0
MOVL C01115 V=800.0 PL=0
MOVL C01116 V=800.0 PL=0
MOVL C01117 V=800.0 PL=0
MOVL C01118 V=800.0 PL=0
MOVL C01119 V=800.0 PL=0
MOVL C01120 V=800.0 PL=0
MOVL C01121 V=800.0 PL=0
MOVL C01122 V=800.0 PL=0
MOVL C01123 V=800.0 PL=0
MOVL C01124 V=800.0 PL=0
MOVL C01125 V=800.0 PL=0
MOVL C01126 V=800.0 PL=0
MOVL C01127 V=800.0 PL=0
MOVL C01128 V=800.0 PL=0
MOVL C01129 V=800.0 PL=0
MOVL C01130 V=800.0 PL=0
MOVL C01131 V=800.0 PL=0
MOVL C01132 V=800.0 PL=0
MOVL C01133 V=800.0 PL=0
MOVL C01134 V=800.0 PL=0
MOVL C01135 V=800.0 PL=0
MOVL C01136 V=800.0 PL=0
MOVL C01137 V=800.0 PL=0
MOVL C01138 V=800.0 PL=0
MOVL C01139 V=800.0 PL=0
MOVL C01140 V=800.0 PL=0
MOVL C01141 V=800.0 PL=0
MOVL C01142 V=800.0 PL=0
MOVL C01143 V=800.0 PL=0
MOVL C01144 V=800.0 PL=0
MOVL C01145 V=800.0 PL=0
MOVL C01146 V=800.0 PL=0
MOVL C01147 V=800.0 PL=0
MOVL C01148 V=800.0 PL=0
MOVL C01149 V=800.0 PL=0
MOVL C01150 V=800.0 PL=0
MOVL C01151 V=800.0 PL=0
MOVL C01152 V=800.0 PL=0
MOVL C01153 V=800.0 PL=0
MOVL C01154 V=800.0 PL=0
MOVL C01155 V=800.0 PL=0
MOVL C01156 V=800.0 PL=0
MOVL C01157 V=800.0 PL=0
MOVL C01158 V=800.0 PL=0
MOVL C01159 V=800.0 PL=0
MOVL C01160 V=800.0 PL=0
MOVL C01161 V=800.0 PL=0
MOVL C01162 V=800.0 PL=0
MOVL C01163 V=800.0 PL=0
MOVL C01164 V=800.0 PL=0
MOVL C01165 V=800.0 PL=0
MOVL C01166 V=800.0 PL=0
MOVL C01167 V=800.0 PL=0
MOVL C01168 V=800.0 PL=0
MOVL C01169 V=800.0 PL=0
MOVL C01170 V=800.0 PL=0
MOVL C01171 V=800.0 PL=0
MOVL C01172 V=800.0 PL=0
MOVL C01173 V=800.0 PL=0
MOVL C01174 V=800.0 PL=0
MOVL C01175 V=800.0 PL=0
MOVL C01176 V=800.0 PL=0
MOVL C01177 V=800.0 PL=0
MOVL C01178 V=800.0 PL=0
MOVL C01179 V=800.0 PL=0
MOVL C01180 V=800.0 PL=0
MOVL C01181 V=800.0 PL=0
MOVL C01182 V=800.0 PL=0
MOVL C01183 V=800.0 PL=0
MOVL C01184 V=800.0 PL=0
MOVL C01185 V=800.0 PL=0
MOVL C01186 V=800.0 PL=0
MOVL C01187 V=800.0 PL=0
MOVL C01188 V=800.0 PL=0
MOVL C01189 V=800.0 PL=0
MOVL C01190 V=800.0 PL=0
MOVL C01191 V=800.0 PL=0
MOVL C01192 V=800.0 PL=0
MOVL C01193 V=800.0 PL=0
MOVL C01194 V=800.0 PL=0
MOVL C01195 V=800.0 PL=0
MOVL C01196 V=800.0 PL=0
MOVL C01197 V=800.0 PL=0
MOVL C01198 V=800.0 PL=0
MOVL C01199 V=800.0 PL=0
MOVL C01200 V=800.0 PL=0
MOVL C01201 V=800.0 PL=0
MOVL C01202 V=800.0 PL=0
MOVL C01203 V=800.0 PL=0
MOVL C01204 V=800.0 PL=0
MOVL C01205 V=800.0 PL=0
MOVL C01206 V=800.0 PL=0
MOVL C01207 V=800.0 PL=0
MOVL C01208 V=800.0 PL=0
MOVL C01209 V=800.0 PL=0
MOVL C01210 V=800.0 PL=0
MOVL C01211 V=800.0 PL=0
MOVL C01212 V=800.0 PL=0
MOVL C01213 V=800.0 PL=0
MOVL C01214 V=800.0 PL=0
MOVL C01215 V=800.0 PL=0
MOVL C01216 V=800.0 PL=0
MOVL C01217 V=800.0 PL=0
MOVL C01218 V=800.0 PL=0
MOVL C01219 V=800.0 PL=0
MOVL C01220 V=800.0 PL=0
MOVL C01221 V=800.0 PL=0
MOVL C01222 V=800.0 PL=0
MOVL C01223 V=800.0 PL=0
MOVL C01224 V=800.0 PL=0
MOVL C01225 V=800.0 PL=0
MOVL C01226 V=800.0 PL=0
MOVL C01227 V=800.0 PL=0
MOVL C01228 V=800.0 PL=0
MOVL C01229 V=800.0 PL=0
MOVL C01230 V=800.0 PL=0
MOVL C01231 V=800.0 PL=0
MOVL C01232 V=800.0 PL=0
MOVL C01233 V=800.0 PL=0
MOVL C01234 V=800.0 PL=0
MOVL C01235 V=800.0 PL=0
MOVL C01236 V=800.0 PL=0
MOVL C01237 V=800.0 PL=0
MOVL C01238 V=800.0 PL=0
MOVL C01239 V=800.0 PL=0
MOVL C01240 V=800.0 PL=0
MOVL C01241 V=800.0 PL=0
MOVL C01242 V=800.0 PL=0
MOVL C01243 V=800.0 PL=0
MOVL C01244 V=800.0 PL=0
MOVL C01245 V=800.0 PL=0
MOVL C01246 V=800.0 PL=0
MOVL C01247 V=800.0 PL=0
MOVL C01248 V=800.0 PL=0
MOVL C01249 V=800.0 PL=0
MOVL C01250 V=800.0 PL=0
MOVL C01251 V=800.0 PL=0
MOVL C01252 V=800.0 PL=0
MOVL C01253 V=800.0 PL=0
MOVL C01254 V=800.0 PL=0
MOVL C01255 V=800.0 PL=0
MOVL C01256 V=800.0 PL=0
MOVL C01257 V=800.0 PL=0
MOVL C01258 V=800.0 PL=0
MOVL C01259 V=800.0 PL=0
MOVL C01260 V=800.0 PL=0
MOVL C01261 V=800.0 PL=0
MOVL C01262 V=800.0 PL=0
MOVL C01263 V=800.0 PL=0
MOVL C01264 V=800.0 PL=0
MOVL C01265 V=800.0 PL=0
MOVL C01266 V=800.0 PL=0
MOVL C01267 V=800.0 PL=0
MOVL C01268 V=800.0 PL=0
MOVL C01269 V=800.0 PL=0
MOVL C01270 V=800.0 PL=0
MOVL C01271 V=800.0 PL=0
MOVL C01272 V=800.0 PL=0
MOVL C01273 V=800.0 PL=0
MOVL C01274 V=800.0 PL=0
MOVL C01275 V=800.0 PL=0
MOVL C01276 V=800.0 PL=0
MOVL C01277 V=800.0 PL=0
MOVL C01278 V=800.0 PL=0
MOVL C01279 V=800.0 PL=0
MOVL C01280 V=800.0 PL=0
MOVL C01281 V=800.0 PL=0
MOVL C01282 V=800.0 PL=0
MOVL C01283 V=800.0 PL=0
MOVL C01284 V=800.0 PL=0
MOVL C01285 V=800.0 PL=0
MOVL C01286 V=800.0 PL=0
MOVL C01287 V=800.0 PL=0
MOVL C01288 V=800.0 PL=0
MOVL C01289 V=800.0 PL=0
MOVL C01290 V=800.0 PL=0
MOVL C01291 V=800.0 PL=0
MOVL C01292 V=800.0 PL=0
MOVL C01293 V=800.0 PL=0
MOVL C01294 V=800.0 PL=0
MOVL C01295 V=800.0 PL=0
MOVL C01296 V=800.0 PL=0
MOVL C01297 V=800.0 PL=0
MOVL C01298 V=800.0 PL=0
MOVL C01299 V=800.0 PL=0
MOVL C01300 V=800.0 PL=0
MOVL C01301 V=800.0 PL=0
MOVL C01302 V=800.0 PL=0
MOVL C01303 V=800.0 PL=0
MOVL C01304 V=800.0 PL=0
MOVL C01305 V=800.0 PL=0
MOVL C01306 V=800.0 PL=0
MOVL C01307 V=800.0 PL=0
MOVL C01308 V=800.0 PL=0
MOVL C01309 V=800.0 PL=0
MOVL C01310 V=800.0 PL=0
MOVL C01311 V=800.0 PL=0
MOVL C01312 V=800.0 PL=0
MOVL C01313 V=800.0 PL=0
MOVL C01314 V=800.0 PL=0
MOVL C01315 V=800.0 PL=0
MOVL C01316 V=800.0 PL=0
MOVL C01317 V=800.0 PL=0
MOVL C01318 V=800.0 PL=0
MOVL C01319 V=800.0 PL=0
MOVL C01320 V=800.0 PL=0
MOVL C01321 V=800.0 PL=0
MOVL C01322 V=800.0 PL=0
MOVL C01323 V=800.0 PL=0
MOVL C01324 V=800.0 PL=0
MOVL C01325 V=800.0 PL=0
MOVL C01326 V=800.0 PL=0
MOVL C01327 V=800.0 PL=0
MOVL C01328 V=800.0 PL=0
MOVL C01329 V=800.0 PL=0
MOVL C01330 V=800.0 PL=0
MOVL C01331 V=800.0 PL=0
MOVL C01332 V=800.0 PL=0
MOVL C01333 V=800.0 PL=0
MOVL C01334 V=800.0 PL=0
MOVL C01335 V=800.0 PL=0
MOVL C01336 V=800.0 PL=0
MOVL C01337 V=800.0 PL=0
MOVL C01338 V=800.0 PL=0
MOVL C01339 V=800.0 PL=0
MOVL C01340 V=800.0 PL=0
MOVL C01341 V=800.0 PL=0
MOVL C01342 V=800.0 PL=0
MOVL C01343 V=800.0 PL=0
MOVL C01344 V=800.0 PL=0
MOVL C01345 V=800.0 PL=0
MOVL C01346 V=800.0 PL=0
MOVL C01347 V=800.0 PL=0
MOVL C01348 V=800.0 PL=0
MOVL C01349 V=800.0 PL=0
MOVL C01350 V=800.0 PL=0
MOVL C01351 V=800.0 PL=0
MOVL C01352 V=800.0 PL=0
MOVL C01353 V=800.0 PL=0
MOVL C01354 V=800.0 PL=0
MOVL C01355 V=800.0 PL=0
MOVL C01356 V=800.0 PL=0
MOVL C01357 V=800.0 PL=0
MOVL C01358 V=800.0 PL=0
MOVL C01359 V=800.0 PL=0
MOVL C01360 V=800.0 PL=0
MOVL C01361 V=800.0 PL=0
MOVL C01362 V=800.0 PL=0
MOVL C01363 V=800.0 PL=0
MOVL C01364 V=800.0 PL=0
MOVL C01365 V=800.0 PL=0
MOVL C01366 V=800.0 PL=0
MOVL C01367 V=800.0 PL=0
MOVL C01368 V=800.0 PL=0
MOVL C01369 V=800.0 PL=0
MOVL C01370 V=800.0 PL=0
MOVL C01371 V=800.0 PL=0
MOVL C01372 V=800.0 PL=0
MOVL C01373 V=800.0 PL=0
MOVL C01374 V=800.0 PL=0
MOVL C01375 V=800.0 PL=0
MOVL C01376 V=800.0 PL=0
MOVL C01377 V=800.0 PL=0
MOVL C01378 V=800.0 PL=0
MOVL C01379 V=800.0 PL=0
MOVL C01380 V=800.0 PL=0
MOVL C01381 V=800.0 PL=0
MOVL C01382 V=800.0 PL=0
MOVL C01383 V=800.0 PL=0
MOVL C01384 V=800.0 PL=0
MOVL C01385 V=800.0 PL=0
MOVL C01386 V=800.0 PL=0
MOVL C01387 V=800.0 PL=0
MOVL C01388 V=800.0 PL=0
MOVL C01389 V=800.0 PL=0
MOVL C01390 V=800.0 PL=0
MOVL C01391 V=800.0 PL=0
MOVL C01392 V=800.0 PL=0
MOVL C01393 V=800.0 PL=0
MOVL C01394 V=800.0 PL=0
MOVL C01395 V=800.0 PL=0
MOVL C01396 V=800.0 PL=0
MOVL C01397 V=800.0 PL=0
MOVL C01398 V=800.0 PL=0
MOVL C01399 V=800.0 PL=0
MOVL C01400 V=800.0 PL=0
MOVL C01401 V=800.0 PL=0
MOVL C01402 V=800.0 PL=0
MOVL C01403 V=800.0 PL=0
MOVL C01404 V=800.0 PL=0
MOVL C01405 V=800.0 PL=0
MOVL C01406 V=800.0 PL=0
MOVL C01407 V=800.0 PL=0
MOVL C01408 V=800.0 PL=0
MOVL C01409 V=800.0 PL=0
MOVL C01410 V=800.0 PL=0
MOVL C01411 V=800.0 PL=0
MOVL C01412 V=800.0 PL=0
MOVL C01413 V=800.0 PL=0
MOVL C01414 V=800.0 PL=0
MOVL C01415 V=800.0 PL=0
MOVL C01416 V=800.0 PL=0
MOVL C01417 V=800.0 PL=0
MOVL C01418 V=800.0 PL=0
MOVL C01419 V=800.0 PL=0
MOVL C01420 V=800.0 PL=0
MOVL C01421 V=800.0 PL=0
MOVL C01422 V=800.0 PL=0
MOVL C01423 V=800.0 PL=0
MOVL C01424 V=800.0 PL=0
MOVL C01425 V=800.0 PL=0
MOVL C01426 V=800.0 PL=0
MOVL C01427 V=800.0 PL=0
MOVL C01428 V=800.0 PL=0
MOVL C01429 V=800.0 PL=0
MOVL C01430 V=800.0 PL=0
MOVL C01431 V=800.0 PL=0
MOVL C01432 V=800.0 PL=0
MOVL C01433 V=800.0 PL=0
MOVL C01434 V=800.0 PL=0
MOVL C01435 V=800.0 PL=0
MOVL C01436 V=800.0 PL=0
MOVL C01437 V=800.0 PL=0
MOVL C01438 V=800.0 PL=0
MOVL C01439 V=800.0 PL=0
MOVL C01440 V=800.0 PL=0
MOVL C01441 V=800.0 PL=0
MOVL C01442 V=800.0 PL=0
MOVL C01443 V=800.0 PL=0
MOVL C01444 V=800.0 PL=0
MOVL C01445 V=800.0 PL=0
MOVL C01446 V=800.0 PL=0
MOVL C01447 V=800.0 PL=0
MOVL C01448 V=800.0 PL=0
MOVL C01449 V=800.0 PL=0
MOVL C01450 V=800.0 PL=0
MOVL C01451 V=800.0 PL=0
MOVL C01452 V=800.0 PL=0
MOVL C01453 V=800.0 PL=0
MOVL C01454 V=800.0 PL=0
MOVL C01455 V=800.0 PL=0
MOVL C01456 V=800.0 PL=0
MOVL C01457 V=800.0 PL=0
MOVL C01458 V=800.0 PL=0
MOVL C01459 V=800.0 PL=0
MOVL C01460 V=800.0 PL=0
MOVL C01461 V=800.0 PL=0
MOVL C01462 V=800.0 PL=0
MOVL C01463 V=800.0 PL=0
MOVL C01464 V=800.0 PL=0
MOVL C01465 V=800.0 PL=0
MOVL C01466 V=800.0 PL=0
MOVL C01467 V=800.0 PL=0
MOVL C01468 V=800.0 PL=0
MOVL C01469 V=800.0 PL=0
MOVL C01470 V=800.0 PL=0
MOVL C01471 V=800.0 PL=0
MOVL C01472 V=800.0 PL=0
MOVL C01473 V=800.0 PL=0
MOVL C01474 V=800.0 PL=0
MOVL C01475 V=800.0 PL=0
MOVL C01476 V=800.0 PL=0
MOVL C01477 V=800.0 PL=0
MOVL C01478 V=800.0 PL=0
MOVL C01479 V=800.0 PL=0
MOVL C01480 V=800.0 PL=0
MOVL C01481 V=800.0 PL=0
MOVL C01482 V=800.0 PL=0
MOVL C01483 V=800.0 PL=0
MOVL C01484 V=800.0 PL=0
MOVL C01485 V=800.0 PL=0
MOVL C01486 V=800.0 PL=0
MOVL C01487 V=800.0 PL=0
MOVL C01488 V=800.0 PL=0
MOVL C01489 V=800.0 PL=0
MOVL C01490 V=800.0 PL=0
MOVL C01491 V=800.0 PL=0
MOVL C01492 V=800.0 PL=0
MOVL C01493 V=800.0 PL=0
MOVL C01494 V=800.0 PL=0
MOVL C01495 V=800.0 PL=0
MOVL C01496 V=800.0 PL=0
MOVL C01497 V=800.0 PL=0
MOVL C01498 V=800.0 PL=0
MOVL C01499 V=800.0 PL=0
MOVL C01500 V=800.0 PL=0
MOVL C01501 V=800.0 PL=0
MOVL C01502 V=800.0 PL=0
MOVL C01503 V=800.0 PL=0
MOVL C01504 V=800.0 PL=0
MOVL C01505 V=800.0 PL=0
MOVL C01506 V=800.0 PL=0
MOVL C01507 V=800.0 PL=0
MOVL C01508 V=800.0 PL=0
MOVL C01509 V=800.0 PL=0
MOVL C01510 V=800.0 PL=0
MOVL C01511 V=800.0 PL=0
MOVL C01512 V=800.0 PL=0
MOVL C01513 V=800.0 PL=0
MOVL C01514 V=800.0 PL=0
MOVL C01515 V=800.0 PL=0
MOVL C01516 V=800.0 PL=0
MOVL C01517 V=800.0 PL=0
MOVL C01518 V=800.0 PL=0
MOVL C01519 V=800.0 PL=0
MOVL C01520 V=800.0 PL=0
MOVL C01521 V=800.0 PL=0
MOVL C01522 V=800.0 PL=0
MOVL C01523 V=800.0 PL=0
MOVL C01524 V=800.0 PL=0
MOVL C01525 V=800.0 PL=0
MOVL C01526 V=800.0 PL=0
MOVL C01527 V=800.0 PL=0
MOVL C01528 V=800.0 PL=0
MOVL C01529 V=800.0 PL=0
MOVL C01530 V=800.0 PL=0
MOVL C01531 V=800.0 PL=0
MOVL C01532 V=800.0 PL=0
MOVL C01533 V=800.0 PL=0
MOVL C01534 V=800.0 PL=0
MOVL C01535 V=800.0 PL=0
MOVL C01536 V=800.0 PL=0
MOVL C01537 V=800.0 PL=0
MOVL C01538 V=800.0 PL=0
MOVL C01539 V=800.0 PL=0
MOVL C01540 V=800.0 PL=0
MOVL C01541 V=800.0 PL=0
MOVL C01542 V=800.0 PL=0
MOVL C01543 V=800.0 PL=0
MOVL C01544 V=800.0 PL=0
MOVL C01545 V=800.0 PL=0
MOVL C01546 V=800.0 PL=0
MOVL C01547 V=800.0 PL=0
MOVL C01548 V=800.0 PL=0
MOVL C01549 V=800.0 PL=0
MOVL C01550 V=800.0 PL=0
MOVL C01551 V=800.0 PL=0
MOVL C01552 V=800.0 PL=0
MOVL C01553 V=800.0 PL=0
MOVL C01554 V=800.0 PL=0
MOVL C01555 V=800.0 PL=0
MOVL C01556 V=800.0 PL=0
MOVL C01557 V=800.0 PL=0
MOVL C01558 V=800.0 PL=0
MOVL C01559 V=800.0 PL=0
MOVL C01560 V=800.0 PL=0
MOVL C01561 V=800.0 PL=0
MOVL C01562 V=800.0 PL=0
MOVL C01563 V=800.0 PL=0
MOVL C01564 V=800.0 PL=0
MOVL C01565 V=800.0 PL=0
MOVL C01566 V=800.0 PL=0
MOVL C01567 V=800.0 PL=0
MOVL C01568 V=800.0 PL=0
MOVL C01569 V=800.0 PL=0
MOVL C01570 V=800.0 PL=0
MOVL C01571 V=800.0 PL=0
MOVL C01572 V=800.0 PL=0
MOVL C01573 V=800.0 PL=0
MOVL C01574 V=800.0 PL=0
MOVL C01575 V=800.0 PL=0
MOVL C01576 V=800.0 PL=0
MOVL C01577 V=800.0 PL=0
MOVL C01578 V=800.0 PL=0
MOVL C01579 V=800.0 PL=0
MOVL C01580 V=800.0 PL=0
MOVL C01581 V=800.0 PL=0
MOVL C01582 V=800.0 PL=0
MOVL C01583 V=800.0 PL=0
MOVL C01584 V=800.0 PL=0
MOVL C01585 V=800.0 PL=0
MOVL C01586 V=800.0 PL=0
MOVL C01587 V=800.0 PL=0
MOVL C01588 V=800.0 PL=0
MOVL C01589 V=800.0 PL=0
MOVL C01590 V=800.0 PL=0
MOVL C01591 V=800.0 PL=0
MOVL C01592 V=800.0 PL=0
MOVL C01593 V=800.0 PL=0
MOVL C01594 V=800.0 PL=0
MOVL C01595 V=800.0 PL=0
MOVL C01596 V=800.0 PL=0
MOVL C01597 V=800.0 PL=0
MOVL C01598 V=800.0 PL=0
MOVL C01599 V=800.0 PL=0
MOVL C01600 V=800.0 PL=0
MOVL C01601 V=800.0 PL=0
MOVL C01602 V=800.0 PL=0
MOVL C01603 V=800.0 PL=0
MOVL C01604 V=800.0 PL=0
MOVL C01605 V=800.0 PL=0
MOVL C01606 V=800.0 PL=0
MOVL C01607 V=800.0 PL=0
MOVL C01608 V=800.0 PL=0
MOVL C01609 V=800.0 PL=0
MOVL C01610 V=800.0 PL=0
MOVL C01611 V=800.0 PL=0
MOVL C01612 V=800.0 PL=0
MOVL C01613 V=800.0 PL=0
MOVL C01614 V=800.0 PL=0
MOVL C01615 V=800.0 PL=0
MOVL C01616 V=800.0 PL=0
MOVL C01617 V=800.0 PL=0
MOVL C01618 V=800.0 PL=0
MOVL C01619 V=800.0 PL=0
MOVL C01620 V=800.0 PL=0
MOVL C01621 V=800.0 PL=0
MOVL C01622 V=800.0 PL=0
MOVL C01623 V=800.0 PL=0
MOVL C01624 V=800.0 PL=0
MOVL C01625 V=800.0 PL=0
MOVL C01626 V=800.0 PL=0
MOVL C01627 V=800.0 PL=0
MOVL C01628 V=800.0 PL=0
MOVL C01629 V=800.0 PL=0
MOVL C01630 V=800.0 PL=0
MOVL C01631 V=800.0 PL=0
MOVL C01632 V=800.0 PL=0
MOVL C01633 V=800.0 PL=0
MOVL C01634 V=800.0 PL=0
MOVL C01635 V=800.0 PL=0
MOVL C01636 V=800.0 PL=0
MOVL C01637 V=800.0 PL=0
MOVL C01638 V=800.0 PL=0
MOVL C01639 V=800.0 PL=0
MOVL C01640 V=800.0 PL=0
MOVL C01641 V=800.0 PL=0
MOVL C01642 V=800.0 PL=0
MOVL C01643 V=800.0 PL=0
MOVL C01644 V=800.0 PL=0
MOVL C01645 V=800.0 PL=0
MOVL C01646 V=800.0 PL=0
MOVL C01647 V=800.0 PL=0
MOVL C01648 V=800.0 PL=0
MOVL C01649 V=800.0 PL=0
MOVL C01650 V=800.0 PL=0
MOVL C01651 V=800.0 PL=0
MOVL C01652 V=800.0 PL=0
MOVL C01653 V=800.0 PL=0
MOVL C01654 V=800.0 PL=0
MOVL C01655 V=800.0 PL=0
MOVL C01656 V=800.0 PL=0
MOVL C01657 V=800.0 PL=0
MOVL C01658 V=800.0 PL=0
MOVL C01659 V=800.0 PL=0
MOVL C01660 V=800.0 PL=0
MOVL C01661 V=800.0 PL=0
MOVL C01662 V=800.0 PL=0
MOVL C01663 V=800.0 PL=0
MOVL C01664 V=800.0 PL=0
MOVL C01665 V=800.0 PL=0
MOVL C01666 V=800.0 PL=0
MOVL C01667 V=800.0 PL=0
MOVL C01668 V=800.0 PL=0
MOVL C01669 V=800.0 PL=0
MOVL C01670 V=800.0 PL=0
MOVL C01671 V=800.0 PL=0
MOVL C01672 V=800.0 PL=0
MOVL C01673 V=800.0 PL=0
MOVL C01674 V=800.0 PL=0
MOVL C01675 V=800.0 PL=0
MOVL C01676 V=800.0 PL=0
MOVL C01677 V=800.0 PL=0
MOVL C01678 V=800.0 PL=0
MOVL C01679 V=800.0 PL=0
MOVL C01680 V=800.0 PL=0
MOVL C01681 V=800.0 PL=0
MOVL C01682 V=800.0 PL=0
MOVL C01683 V=800.0 PL=0
MOVL C01684 V=800.0 PL=0
MOVL C01685 V=800.0 PL=0
MOVL C01686 V=800.0 PL=0
MOVL C01687 V=800.0 PL=0
MOVL C01688 V=800.0 PL=0
MOVL C01689 V=800.0 PL=0
MOVL C01690 V=800.0 PL=0
MOVL C01691 V=800.0 PL=0
MOVL C01692 V=800.0 PL=0
MOVL C01693 V=800.0 PL=0
MOVL C01694 V=800.0 PL=0
MOVL C01695 V=800.0 PL=0
MOVL C01696 V=800.0 PL=0
MOVL C01697 V=800.0 PL=0
MOVL C01698 V=800.0 PL=0
MOVL C01699 V=800.0 PL=0
MOVL C01700 V=800.0 PL=0
MOVL C01701 V=800.0 PL=0
MOVL C01702 V=800.0 PL=0
MOVL C01703 V=800.0 PL=0
MOVL C01704 V=800.0 PL=0
MOVL C01705 V=800.0 PL=0
MOVL C01706 V=800.0 PL=0
MOVL C01707 V=800.0 PL=0
MOVL C01708 V=800.0 PL=0
MOVL C01709 V=800.0 PL=0
MOVL C01710 V=800.0 PL=0
MOVL C01711 V=800.0 PL=0
MOVL C01712 V=800.0 PL=0
MOVL C01713 V=800.0 PL=0
MOVL C01714 V=800.0 PL=0
MOVL C01715 V=800.0 PL=0
MOVL C01716 V=800.0 PL=0
MOVL C01717 V=800.0 PL=0
MOVL C01718 V=800.0 PL=0
MOVL C01719 V=800.0 PL=0
MOVL C01720 V=800.0 PL=0
MOVL C01721 V=800.0 PL=0
MOVL C01722 V=800.0 PL=0
MOVL C01723 V=800.0 PL=0
MOVL C01724 V=800.0 PL=0
MOVL C01725 V=800.0 PL=0
MOVL C01726 V=800.0 PL=0
MOVL C01727 V=800.0 PL=0
MOVL C01728 V=800.0 PL=0
MOVL C01729 V=800.0 PL=0
MOVL C01730 V=800.0 PL=0
MOVL C01731 V=800.0 PL=0
MOVL C01732 V=800.0 PL=0
MOVL C01733 V=800.0 PL=0
MOVL C01734 V=800.0 PL=0
MOVL C01735 V=800.0 PL=0
MOVL C01736 V=800.0 PL=0
MOVL C01737 V=800.0 PL=0
MOVL C01738 V=800.0 PL=0
MOVL C01739 V=800.0 PL=0
MOVL C01740 V=800.0 PL=0
MOVL C01741 V=800.0 PL=0
MOVL C01742 V=800.0 PL=0
MOVL C01743 V=800.0 PL=0
MOVL C01744 V=800.0 PL=0
MOVL C01745 V=800.0 PL=0
MOVL C01746 V=800.0 PL=0
MOVL C01747 V=800.0 PL=0
MOVL C01748 V=800.0 PL=0
MOVL C01749 V=800.0 PL=0
MOVL C01750 V=800.0 PL=0
MOVL C01751 V=800.0 PL=0
MOVL C01752 V=800.0 PL=0
MOVL C01753 V=800.0 PL=0
MOVL C01754 V=800.0 PL=0
MOVL C01755 V=800.0 PL=0
MOVL C01756 V=800.0 PL=0
MOVL C01757 V=800.0 PL=0
MOVL C01758 V=800.0 PL=0
MOVL C01759 V=800.0 PL=0
MOVL C01760 V=800.0 PL=0
MOVL C01761 V=800.0 PL=0
MOVL C01762 V=800.0 PL=0
MOVL C01763 V=800.0 PL=0
MOVL C01764 V=800.0 PL=0
MOVL C01765 V=800.0 PL=0
MOVL C01766 V=800.0 PL=0
MOVL C01767 V=800.0 PL=0
MOVL C01768 V=800.0 PL=0
MOVL C01769 V=800.0 PL=0
MOVL C01770 V=800.0 PL=0
MOVL C01771 V=800.0 PL=0
MOVL C01772 V=800.0 PL=0
MOVL C01773 V=800.0 PL=0
MOVL C01774 V=800.0 PL=0
MOVL C01775 V=800.0 PL=0
MOVL C01776 V=800.0 PL=0
MOVL C01777 V=800.0 PL=0
MOVL C01778 V=800.0 PL=0
MOVL C01779 V=800.0 PL=0
MOVL C01780 V=800.0 PL=0
MOVL C01781 V=800.0 PL=0
MOVL C01782 V=800.0 PL=0
MOVL C01783 V=800.0 PL=0
MOVL C01784 V=800.0 PL=0
MOVL C01785 V=800.0 PL=0
MOVL C01786 V=800.0 PL=0
MOVL C01787 V=800.0 PL=0
MOVL C01788 V=800.0 PL=0
MOVL C01789 V=800.0 PL=0
MOVL C01790 V=800.0 PL=0
MOVL C01791 V=800.0 PL=0
MOVL C01792 V=800.0 PL=0
MOVL C01793 V=800.0 PL=0
MOVL C01794 V=800.0 PL=0
MOVL C01795 V=800.0 PL=0
MOVL C01796 V=800.0 PL=0
MOVL C01797 V=800.0 PL=0
MOVL C01798 V=800.0 PL=0
MOVL C01799 V=800.0 PL=0
MOVL C01800 V=800.0 PL=0
MOVL C01801 V=800.0 PL=0
MOVL C01802 V=800.0 PL=0
MOVL C01803 V=800.0 PL=0
MOVL C01804 V=800.0 PL=0
MOVL C01805 V=800.0 PL=0
MOVL C01806 V=800.0 PL=0
MOVL C01807 V=800.0 PL=0
MOVL C01808 V=800.0 PL=0
MOVL C01809 V=800.0 PL=0
MOVL C01810 V=800.0 PL=0
MOVL C01811 V=800.0 PL=0
MOVL C01812 V=800.0 PL=0
MOVL C01813 V=800.0 PL=0
MOVL C01814 V=800.0 PL=0
MOVL C01815 V=800.0 PL=0
MOVL C01816 V=800.0 PL=0
MOVL C01817 V=800.0 PL=0
MOVL C01818 V=800.0 PL=0
MOVL C01819 V=800.0 PL=0
MOVL C01820 V=800.0 PL=0
MOVL C01821 V=800.0 PL=0
MOVL C01822 V=800.0 PL=0
MOVL C01823 V=800.0 PL=0
MOVL C01824 V=800.0 PL=0
MOVL C01825 V=800.0 PL=0
MOVL C01826 V=800.0 PL=0
MOVL C01827 V=800.0 PL=0
MOVL C01828 V=800.0 PL=0
MOVL C01829 V=800.0 PL=0
MOVL C01830 V=800.0 PL=0
MOVL C01831 V=800.0 PL=0
MOVL C01832 V=800.0 PL=0
MOVL C01833 V=800.0 PL=0
MOVL C01834 V=800.0 PL=0
MOVL C01835 V=800.0 PL=0
MOVL C01836 V=800.0 PL=0
MOVL C01837 V=800.0 PL=0
MOVL C01838 V=800.0 PL=0
MOVL C01839 V=800.0 PL=0
MOVL C01840 V=800.0 PL=0
MOVL C01841 V=800.0 PL=0
MOVL C01842 V=800.0 PL=0
MOVL C01843 V=800.0 PL=0
MOVL C01844 V=800.0 PL=0
MOVL C01845 V=800.0 PL=0
MOVL C01846 V=800.0 PL=0
MOVL C01847 V=800.0 PL=0
MOVL C01848 V=800.0 PL=0
MOVL C01849 V=800.0 PL=0
MOVL C01850 V=800.0 PL=0
MOVL C01851 V=800.0 PL=0
MOVL C01852 V=800.0 PL=0
MOVL C01853 V=800.0 PL=0
MOVL C01854 V=800.0 PL=0
MOVL C01855 V=800.0 PL=0
MOVL C01856 V=800.0 PL=0
MOVL C01857 V=800.0 PL=0
MOVL C01858 V=800.0 PL=0
MOVL C01859 V=800.0 PL=0
MOVL C01860 V=800.0 PL=0
MOVL C01861 V=800.0 PL=0
MOVL C01862 V=800.0 PL=0
MOVL C01863 V=800.0 PL=0
MOVL C01864 V=800.0 PL=0
MOVL C01865 V=800.0 PL=0
MOVL C01866 V=800.0 PL=0
MOVL C01867 V=800.0 PL=0
MOVL C01868 V=800.0 PL=0
MOVL C01869 V=800.0 PL=0
MOVL C01870 V=800.0 PL=0
MOVL C01871 V=800.0 PL=0
MOVL C01872 V=800.0 PL=0
MOVL C01873 V=800.0 PL=0
MOVL C01874 V=800.0 PL=0
MOVL C01875 V=800.0 PL=0
MOVL C01876 V=800.0 PL=0
MOVL C01877 V=800.0 PL=0
MOVL C01878 V=800.0 PL=0
MOVL C01879 V=800.0 PL=0
MOVL C01880 V=800.0 PL=0
MOVL C01881 V=800.0 PL=0
MOVL C01882 V=800.0 PL=0
MOVL C01883 V=800.0 PL=0
MOVL C01884 V=800.0 PL=0
MOVL C01885 V=800.0 PL=0
MOVL C01886 V=800.0 PL=0
MOVL C01887 V=800.0 PL=0
MOVL C01888 V=800.0 PL=0
MOVL C01889 V=800.0 PL=0
MOVL C01890 V=800.0 PL=0
MOVL C01891 V=800.0 PL=0
MOVL C01892 V=800.0 PL=0
MOVL C01893 V=800.0 PL=0
MOVL C01894 V=800.0 PL=0
MOVL C01895 V=800.0 PL=0
MOVL C01896 V=800.0 PL=0
MOVL C01897 V=800.0 PL=0
MOVL C01898 V=800.0 PL=0
MOVL C01899 V=800.0 PL=0
MOVL C01900 V=800.0 PL=0
MOVL C01901 V=800.0 PL=0
MOVL C01902 V=800.0 PL=0
MOVL C01903 V=800.0 PL=0
MOVL C01904 V=800.0 PL=0
MOVL C01905 V=800.0 PL=0
MOVL C01906 V=800.0 PL=0
MOVL C01907 V=800.0 PL=0
MOVL C01908 V=800.0 PL=0
MOVL C01909 V=800.0 PL=0
MOVL C01910 V=800.0 PL=0
MOVL C01911 V=800.0 PL=0
MOVL C01912 V=800.0 PL=0
MOVL C01913 V=800.0 PL=0
MOVL C01914 V=800.0 PL=0
MOVL C01915 V=800.0 PL=0
MOVL C01916 V=800.0 PL=0
MOVL C01917 V=800.0 PL=0
MOVL C01918 V=800.0 PL=0
MOVL C01919 V=800.0 PL=0
MOVL C01920 V=800.0 PL=0
MOVL C01921 V=800.0 PL=0
MOVL C01922 V=800.0 PL=0
MOVL C01923 V=800.0 PL=0
MOVL C01924 V=800.0 PL=0
MOVL C01925 V=800.0 PL=0
MOVL C01926 V=800.0 PL=0
MOVL C01927 V=800.0 PL=0
MOVL C01928 V=800.0 PL=0
MOVL C01929 V=800.0 PL=0
MOVL C01930 V=800.0 PL=0
MOVL C01931 V=800.0 PL=0
MOVL C01932 V=800.0 PL=0
MOVL C01933 V=800.0 PL=0
MOVL C01934 V=800.0 PL=0
MOVL C01935 V=800.0 PL=0
MOVL C01936 V=800.0 PL=0
MOVL C01937 V=800.0 PL=0
MOVL C01938 V=800.0 PL=0
MOVL C01939 V=800.0 PL=0
MOVL C01940 V=800.0 PL=0
MOVL C01941 V=800.0 PL=0
MOVL C01942 V=800.0 PL=0
MOVL C01943 V=800.0 PL=0
MOVL C01944 V=800.0 PL=0
MOVL C01945 V=800.0 PL=0
MOVL C01946 V=800.0 PL=0
MOVL C01947 V=800.0 PL=0
MOVL C01948 V=800.0 PL=0
MOVL C01949 V=800.0 PL=0
MOVL C01950 V=800.0 PL=0
MOVL C01951 V=800.0 PL=0
MOVL C01952 V=800.0 PL=0
MOVL C01953 V=800.0 PL=0
MOVL C01954 V=800.0 PL=0
MOVL C01955 V=800.0 PL=0
MOVL C01956 V=800.0 PL=0
MOVL C01957 V=800.0 PL=0
MOVL C01958 V=800.0 PL=0
MOVL C01959 V=800.0 PL=0
MOVL C01960 V=800.0 PL=0
MOVL C01961 V=800.0 PL=0
MOVL C01962 V=800.0 PL=0
MOVL C01963 V=800.0 PL=0
MOVL C01964 V=800.0 PL=0
MOVL C01965 V=800.0 PL=0
MOVL C01966 V=800.0 PL=0
MOVL C01967 V=800.0 PL=0
MOVL C01968 V=800.0 PL=0
MOVL C01969 V=800.0 PL=0
MOVL C01970 V=800.0 PL=0
MOVL C01971 V=800.0 PL=0
MOVL C01972 V=800.0 PL=0
MOVL C01973 V=800.0 PL=0
MOVL C01974 V=800.0 PL=0
MOVL C01975 V=800.0 PL=0
MOVL C01976 V=800.0 PL=0
MOVL C01977 V=800.0 PL=0
MOVL C01978 V=800.0 PL=0
MOVL C01979 V=800.0 PL=0
MOVL C01980 V=800.0 PL=0
MOVL C01981 V=800.0 PL=0
MOVL C01982 V=800.0 PL=0
MOVL C01983 V=800.0 PL=0
MOVL C01984 V=800.0 PL=0
MOVL C01985 V=800.0 PL=0
MOVL C01986 V=800.0 PL=0
MOVL C01987 V=800.0 PL=0
MOVL C01988 V=800.0 PL=0
MOVL C01989 V=800.0 PL=0
MOVL C01990 V=800.0 PL=0
MOVL C01991 V=800.0 PL=0
MOVL C01992 V=800.0 PL=0
MOVL C01993 V=800.0 PL=0
MOVL C01994 V=800.0 PL=0
MOVL C01995 V=800.0 PL=0
MOVL C01996 V=800.0 PL=0
MOVL C01997 V=800.0 PL=0
MOVL C01998 V=800.0 PL=0
MOVL C01999 V=800.0 PL=0
MOVL C02000 V=800.0 PL=0
MOVL C02001 V=800.0 PL=0
MOVL C02002 V=800.0 PL=0
MOVL C02003 V=800.0 PL=0
MOVL C02004 V=800.0 PL=0
MOVL C02005 V=800.0 PL=0
MOVL C02006 V=800.0 PL=0
MOVL C02007 V=800.0 PL=0
MOVL C02008 V=800.0 PL=0
MOVL C02009 V=800.0 PL=0
MOVL C02010 V=800.0 PL=0
MOVL C02011 V=800.0 PL=0
MOVL C02012 V=800.0 PL=0
MOVL C02013 V=800.0 PL=0
MOVL C02014 V=800.0 PL=0
MOVL C02015 V=800.0 PL=0
MOVL C02016 V=800.0 PL=0
MOVL C02017 V=800.0 PL=0
MOVL C02018 V=800.0 PL=0
MOVL C02019 V=800.0 PL=0
MOVL C02020 V=800.0 PL=0
MOVL C02021 V=800.0 PL=0
MOVL C02022 V=800.0 PL=0
MOVL C02023 V=800.0 PL=0
MOVL C02024 V=800.0 PL=0
MOVL C02025 V=800.0 PL=0
MOVL C02026 V=800.0 PL=0
